END_FUNCTION_BLOCK

// ---- PLC/MAIN.TcPOU
PROGRAM MAIN
VAR
	GetTime: NT_GetTime;
	cpuusage:TC_CpuUsage;
	getLocalAMS: FB_GetLocalAmsNetId;
	ReadSystemInfo:PLC_ReadSymInfo;
	getLatency:TC_SysLatency;
	restartTC:TC_Restart;
	stopTC:TC_Stop;
	configModeTC:TC_Config;
	reqHostName:FB_GetHostName;
	getNetworkadaptors:FB_GetAdaptersInfo;
	getDeviceInfoEx:FB_GetDeviceIdentificationEx;
	
	getLicences:FB_GetLicensesEx;
	
	
	

	oneSec: fb_flasher;
	twoSec: fb_flasher;
	tenSec: fb_flasher;
	oneMSec: fb_flasher;
	hundredMSec: fb_flasher;
	
	pulseoneSec: R_TRIG;
	pulsetwoSec: R_TRIG;
	pulsetenSec: R_TRIG;
	pulseoneMSec: R_TRIG;
	pulsehundredMSec: R_TRIG;
	i: INT;
	nLicPres: UDINT;
	
	oneSecStart:TON;
	
END_VAR

//call PLC data
actPLC();

//call init data for machine
actInit();

//call clock memory
actClockMemory();

//call all diagnostics
actDiag();

//call licence view
actLicenceView();

//call safety main
prgSafetyMain();


//call base machine

//call HMI
//calls logic to drive the HMI
pouHMI();

//call machine base
pouMachine();

//call station 1
//calls motions only associated with station 1
IF System.gSetup.stationEnable[1] THEN pouStation1(); END_IF;

//call station 2
IF System.gSetup.stationEnable[2] THEN pouStation2(); END_IF;

//call station 3
IF System.gSetup.stationEnable[3] THEN pouStation3(); END_IF;

//call station 4
IF System.gSetup.stationEnable[4] THEN pouStation4(); END_IF;

//call station 5
IF System.gSetup.stationEnable[5] THEN pouStation5(); END_IF;

//call station 6
IF System.gSetup.stationEnable[6] THEN pouStation6(); END_IF;

//there are only ever 6 maximum stations

//call logic after station calls for scan after the call of stations
prgAfterStationScan();


//test call for data view
pouDataDisplay();

//call mode rows - call after to use scan logic
prgModeRows();

//call program for machine settings
pouMachineSettings();

//test call for data analyse
prgDataAnaylse();

ACTION actClockMemory:
//clock memory call

//timer call
oneMsec(timeVal:=T#1MS);
System.oneMilliSecond:=oneMSec.q;
pulseoneMSec(CLK:= System.oneMilliSecond);
System.PulseOneMilliSecond := pulseoneMSec.Q;

oneSec(timeVal:=T#1S);
System.OneSecond:=oneSec.q;
pulseoneSec(CLK:= System.OneSecond);
System.PulseOneSecond  := pulseoneSec.Q;

twoSec(timeVal:=T#1S);
System.TwoSecond:=twoSec.q;
pulseTwoSec(CLK:= System.TwoSecond);
System.PulseTwosecond  := pulsetwoSec.Q;

tenSec(timeVal:=T#10S);
System.TenSecond:=tenSec.q;
pulsetenSec(CLK:= System.TenSecond);
System.PulseTenSecond := pulsetenSec.Q;

hundredMSec(timeVal:=T#100MS);
System.hundredMilliSecond:=hundredMSec.q;
pulsehundredMSec(CLK:= System.hundredMilliSecond);
System.PulseHundredMilliSecond := pulsehundredMSec.Q;

oneSecStart(IN:=TRUE);
System.StartPulse:=(oneSecStart.Q);




IF system.thetime.wDay = 28 AND System.thetime.wMonth = 11 THEN
	System.gHappyBirthday := TRUE;
	ELSE
	System.gHappyBirthday := FALSE;
END_IF
END_ACTION

ACTION actDiag:
//call diag blocks
pouDPDiag();
pouEtherCATdiag();
pouPROFINETdiag();
END_ACTION

ACTION actInit:
//block must be called first in scan

//Initalise PLC data for first scan

//activate the first station
IF System.myPlcInfoTask1.FirstCycle THEN
	gHMIData.gActiveStationNumber := 1;
	gHMIData.gStationSelected[1] := TRUE;
	gHMIData.gStationSelected[2] := FALSE;
	gHMIData.gStationSelected[3] := FALSE;
	gHMIData.gStationSelected[4] := FALSE;
	gHMIData.gStationSelected[5] := FALSE;
	gHMIData.gStationSelected[6] := FALSE;
	
	
	//start in manual mode
	S1_Global.station.Data.Manual := TRUE;
	S1_Global.station.Data.AutoCycle := FALSE;
	S1_Global.station.Data.ContCycle := TRUE;
	S1_Global.station.Data.SingleCycle := FALSE;
	
	FC_S1_AssignTaskTimes(iqPartData:=S1_Global.station);
	FC_S2_AssignTaskTimes(iqPartData:=S2_Global.station);
	FC_S3_AssignTaskTimes(iqPartData:=S3_Global.station);
	FC_S4_AssignTaskTimes(iqPartData:=S4_Global.station);
	FC_S5_AssignTaskTimes(iqPartData:=S5_Global.station);
	FC_S6_AssignTaskTimes(iqPartData:=S6_Global.station);
	
	
END_IF

//globals used in future scan(s)
GlobalMessages.gAnyWarnings := FALSE;
GlobalMessages.gAnyFaultMessage := FALSE;

//set other parameters
FC_Setup();
END_ACTION

ACTION actLicenceView:
	//get licence info
	getLicences		(	bExecute:= gLicenceView.tCallUpdateLicenceList,
						tTimeout:=T#10S,
						sNetId:=
					);
	//reset read BOOL
	gLicenceView.tCallUpdateLicenceList := FALSE;
					
gLicenceView.nValidLicences		:=	getLicences.nValidLicenses;
gLicenceView.aValidLicences		:=	getLicences.aValidLicenses;

gLicenceView.nPendingLicences	:=	getLicences.nPendingLicenses;
gLicenceView.aPendingLicences	:=	getLicences.aPendingLicenses;

gLicenceView.nDemoLicences		:=	getLicences.nDemoLicenses;
gLicenceView.aDemoLicences		:=	getLicences.aDemoLicenses;

gLicenceView.nOEMLicences		:=	getLicences.nOemLicenses;
gLicenceView.aOEMLicences		:=	getLicences.aOemLicenses;

gLicenceView.nFailedLicences	:=	getLicences.nFailedLicenses;
gLicenceView.aFailedLicences	:=	getLicences.aFailedLicenses;

gLicenceView.nInvalidLicences	:=	getLicences.nInvalidLicenses;
gLicenceView.aInvalidLicences	:=	getLicences.aInvalidLicenses;

//gLicenceView.maxlicenceIndex := 	gLicenceView.nDemoLicences;
//gLicenceView.tActiveLicenceArray := gLicenceView.ademoLicences[1];


//check if last radio index was changed
IF gLicenceView.licenceType = gLicenceView.tActiveLicenceSelLast THEN
	;
	ELSE
		
	//update list BOOL
	gLicenceView.tCallUpdateLicenceList := TRUE;
	//reset check for next scan
	gLicenceView.tActiveLicenceSelLast :=  gLicenceView.licenceType;
	
END_IF

//assign licence name into array
IF gLicenceView.tCallUpdateLicenceList THEN
	
	//set integer limits for array selection
gLicenceView.tActiveLicenceSel := MAX(gLicenceView.tActiveLicenceSel,1);
gLicenceView.tActiveLicenceSel := MIN(gLicenceView.tActiveLicenceSel,nMaxLicenses);

	
	memset( destAddr:=	ADR(gLicenceView.tActiveLicenceArray),
		 	fillByte:=	16#0,
			n:=			SIZEOF(gLicenceView.tActiveLicenceArray)
			);
	
	memset( destAddr:=	ADR(gLicenceView.tActiveLicenceList),
		 	fillByte:=	16#0,
			n:=			SIZEOF(gLicenceView.tActiveLicenceList)
			);
			
		
	
	
	CASE gLicenceView.licenceType OF
		0:
		gLicenceView.maxlicenceIndex := 	gLicenceView.nValidLicences;
		FOR nLicPres := 1 TO gLicenceView.maxlicenceIndex DO
			gLicenceView.tActiveLicenceList[nLicPres] := gLicenceView.aValidLicences[nLicPres].sLicenseName;
		END_FOR
		
		1:
		gLicenceView.maxlicenceIndex := 	gLicenceView.nPendingLicences;
		FOR nLicPres := 1 TO gLicenceView.maxlicenceIndex DO
			gLicenceView.tActiveLicenceList[nLicPres] := gLicenceView.aPendingLicences[nLicPres].sLicenseName;
		END_FOR
		
		2:
		gLicenceView.maxlicenceIndex := 	gLicenceView.nDemoLicences;
		FOR nLicPres := 1 TO gLicenceView.maxlicenceIndex DO
			gLicenceView.tActiveLicenceList[nLicPres] := gLicenceView.aDemoLicences[nLicPres].sLicenseName;
		END_FOR
		
		3:
		gLicenceView.maxlicenceIndex := 	gLicenceView.nOEMLicences;
		FOR nLicPres := 1 TO gLicenceView.maxlicenceIndex DO
			gLicenceView.tActiveLicenceList[nLicPres] := gLicenceView.aOEMLicences[nLicPres].sLicenseName;
		END_FOR
		
		4:
		gLicenceView.maxlicenceIndex := 	gLicenceView.nFailedLicences;
		FOR nLicPres := 1 TO gLicenceView.maxlicenceIndex DO
			gLicenceView.tActiveLicenceList[nLicPres] := gLicenceView.aFailedLicences[nLicPres].sLicenseName;
		END_FOR
		
		5:
		gLicenceView.maxlicenceIndex := 	gLicenceView.nInvalidLicences;
		FOR nLicPres := 1 TO gLicenceView.maxlicenceIndex DO
			gLicenceView.tActiveLicenceList[nLicPres] := gLicenceView.aInvalidLicences[nLicPres].sLicenseName;
		END_FOR
	
	END_CASE
END_IF

//move data structure into sole struct on HMI
IF gLicenceView.licenceType > 0 THEN

CASE gLicenceView.licenceType OF
	0: 
	//move selected array into viewing arrayh
	gLicenceView.tActiveLicenceArray := gLicenceView.aValidLicences[gLicenceView.tActiveLicenceSel];
	
	1: 
	//move selected array into viewing arrayh
	gLicenceView.tActiveLicenceArray := gLicenceView.aPendingLicences[gLicenceView.tActiveLicenceSel];
	
	2: 
	//move selected array into viewing arrayh
	gLicenceView.tActiveLicenceArray := gLicenceView.aDemoLicences[gLicenceView.tActiveLicenceSel];
	
	3: 
	//move selected array into viewing arrayh
	gLicenceView.tActiveLicenceArray := gLicenceView.aOEMLicences[gLicenceView.tActiveLicenceSel];
	
	4: 
	//move selected array into viewing arrayh
	gLicenceView.tActiveLicenceArray := gLicenceView.aFailedLicences[gLicenceView.tActiveLicenceSel];
	
	5: 
	//move selected array into viewing arrayh
	gLicenceView.tActiveLicenceArray := gLicenceView.aInvalidLicences[gLicenceView.tActiveLicenceSel];
	
END_CASE
END_IF
END_ACTION

ACTION actPLC:
//act call PLC
//get PLC app data
	System.myPlcAppSystemInfo:=TwinCAT_SystemInfoVarList._AppInfo;
	
	//get task info
	System.myPlcInfoTask1 := TwinCAT_SystemInfoVarList._TaskInfo[1];
	
	//move task scan time to memory
	System.ScanTimeReq := UDINT_TO_REAL(System.myPlcInfoTask1.CycleTime);
	System.ScanTimeAct := UDINT_TO_REAL(System.myPlcInfoTask1.LastExecTime);
	
	//scale to correct factor
	System.ScanTimeReq := System.ScanTimeReq / 10000;
	System.ScanTimeAct := System.ScanTimeAct / 10000;
	
	//if the scan time is a new record, then save the scan time and the scan number
	IF System.ScanTimeAct > System.ScanTimeRecord  THEN
		//debug message for new record scan
		System.ScanTimeRecord := System.ScanTimeAct;
		System.ScanTimeRecordScan:= System.myPlcInfoTask1.CycleCount;
	END_IF
	
	//get the local AMS address
	getLocalAMS(	bExecute:=System.myPlcInfoTask1.FirstCycle, 
					tTimeOut:=T#1M
				);
	
	System.AmsNetIdstr:=getLocalAMS.AddrString;
	System.AmsNetIdbytes:=getLocalAMS.AddrBytes;
	
	//get the time
	GetTime(		NETID:='',
					START:=System.OneSecond,
			);
	
	System.thetime:= GetTime.TIMESTR;
	
	//convert timestruct to DT time
	System.timeDT := SYSTEMTIME_TO_DT(TIMESTR:=system.thetime);

	
	//get CPU usage
	cpuusage(	netID:=,
				Start:=System.PulseHundredMilliSecond,
				TMOUT:=T#10S
				);
	System.cpuusageval  := cpuusage.USAGE;
	
	//get symbol count, usage
	ReadSystemInfo( NETID:=,
					Port:=System.myPlcAppSystemInfo.AdsPort,
					Start:=system.OneSecond,
					TMOUT:=T#10S,
					);
	system.symCount:=ReadSystemInfo.SYMCOUNT;
	system.sysSize:=ReadSystemInfo.SYMSIZE;
	
	//get latency
	getLatency(		NETID:=,
					Start:=system.OneSecond,
					TMOUT:=T#10S,
					);
	System.LatencyMicroSec := getLatency.ACTUAL;
	system.MaxLatencyMicroSec := getLatency.MAXIMUM;
	
	//restart TC
	restartTC(		NETID:=,
					Restart:=System.TCRestartReq,
					TMOUT:=T#10S
					);
					
	//stop TC
	stopTC(			NETID:=,
					STOP:=System.TCStopReq,
					TMOUT:=T#10S
					);
					
	//config mode TC
	configModeTC(	NETID:=,
					SET:=System.TCConfigReq,
					TMOUT:=T#10S
					);
				
	//get host name
	reqHostName(	sNetID:=,
					bExecute:=system.TenSecond,
					tTimeout:=T#10S
					);
	System.NThostname := reqHostName.sHostName;
	
	
	//get networkadaptors
	getNetworkadaptors(	sNetID:=,
						bExecute:=system.TenSecond,
						tTimeout:=T#10S,
						);
	System.networkadaptors:=getNetworkadaptors.arrAdapters;
	
	//get Device Infomation
	getDeviceInfoEx(	bExecute := System.sysDeviceUpdate,
						tTimeout := T#10S,
						sNetId:=
					);
					
	System.sysDeviceInfo := getDeviceInfoEx.stDevIdent;
	
	IF gHMIButtons.gAnyMotionButtonPresed THEN gHMIButtons.gAnyMotionButtonPresed := FALSE; END_IF//first scan
END_ACTION

END_PROGRAM

// ---- PLC/FBs/FBs/FB_Flasher.TcPOU
FUNCTION_BLOCK FB_Flasher
VAR
	timON: TON;
	timOFF: TON;

END_VAR

VAR_INPUT
	timeVal:TIME;
	
END_VAR

VAR_OUTPUT
	q:BOOL;

END_VAR

//time on flasher
timON(	IN:= NOT timOFF.Q,
		PT:= timeVal
		);
		
q:= timON.Q;


//time off
timOFF(	IN:= timON.Q,
		PT:= timeVal
		);

END_FUNCTION_BLOCK

// ---- PLC/Safety/prgSafetyMain.TcPOU
PROGRAM prgSafetyMain
VAR
	allowpendantUsage: BOOL; //TRUE if the operator has selected on the HMI to enable the pendant
	runSafeProgram: BOOL; //TRUE to run the safety program
END_VAR



//theme:lOkFAHbeCio

//Main Safety Program Call

//run safety program
IF gHMIButtons.btnReset THEN
	runSafeProgram := TRUE;
END_IF

//add logic TBD to stop safety program

//this send the enable to run the program, should be running all the time in most cases
IF runSafeProgram THEN
	Safety.qInRun := TRUE;
END_IF


//enable pendent logic tbd
allowpendantUsage := FALSE;


//send reset to safety program runtime
IF gHMIButtons.btnReset THEN
	Safety.iResetFBs := TRUE;
	ELSE
	Safety.iResetFBs := FALSE;
END_IF

//to prevent a reset button enabling power devices, have seperate enable fed from HMI
//scan in 0 value
Safety.iEnableSafetyDevicesuint := 0;
IF S1_Global.station.Data.MotionPowerOn AND NOT allowpendantUsage THEN
	//if the station power (or machine power to edit) is on, send value of 1 to enable logic in safety program
	Safety.iEnableSafetyDevicesuint := 1;
END_IF

//pendent enable usage
//scan in 0 value
Safety.iEnablePendantSafetyDevicesuint := 0;
IF allowpendantUsage THEN
	//if the HMI has selected a pendant to use then turn on logic in program
	Safety.iEnablePendantSafetyDevicesuint := 1;
END_IF

END_PROGRAM

// ---- HMI1/Logic/pouHMI.TcPOU
PROGRAM pouHMI
VAR
END_VAR

//all logic to control HMI
prgHMIcontrol();

//control Unit Screen
prgHMIUnits();

//logic for stations
prgHMIstations();

//call to read text lists into PLC memory arrays
prgReadTextList();

//control language Screen
prgHMILanguage();

//axis telegram diag screen
prgHMIaxis();

//lock station logic
actLockStation();

//for Toast-hmi only
actMoveToastHMIData();

ACTION actLockStation:
//lock stations together feedback

IF gHMIButtons.btnLockStation1 THEN gHMIData.gStateLockStation1 := 1; ELSE gHMIData.gStateLockStation1 := 0 ; END_IF
IF gHMIButtons.btnLockStation2 THEN gHMIData.gStateLockStation2 := 1; ELSE gHMIData.gStateLockStation2 := 0 ; END_IF
IF gHMIButtons.btnLockStation3 THEN gHMIData.gStateLockStation3 := 1; ELSE gHMIData.gStateLockStation3 := 0 ; END_IF	
IF gHMIButtons.btnLockStation4 THEN gHMIData.gStateLockStation4 := 1; ELSE gHMIData.gStateLockStation4 := 0 ; END_IF
IF gHMIButtons.btnLockStation5 THEN gHMIData.gStateLockStation5 := 1; ELSE gHMIData.gStateLockStation5 := 0 ; END_IF
IF gHMIButtons.btnLockStation6 THEN gHMIData.gStateLockStation6 := 1; ELSE gHMIData.gStateLockStation6 := 0 ; END_IF
	

//apply locks to stations
S1_Global.station.Data.IsStationLocked	:=	gHMIButtons.btnLockStation1;
S2_Global.station.Data.IsStationLocked	:=	gHMIButtons.btnLockStation2;
S3_Global.station.Data.IsStationLocked	:=	gHMIButtons.btnLockStation3;
S4_Global.station.Data.IsStationLocked	:=	gHMIButtons.btnLockStation4;
S5_Global.station.Data.IsStationLocked	:=	gHMIButtons.btnLockStation5;
S6_Global.station.Data.IsStationLocked	:=	gHMIButtons.btnLockStation6;
END_ACTION

ACTION actMoveToastHMIData:
//move data to new gMHIData to read, not the root for ADS reads

//station selected as BOOL
	gTOASTHMI.gData.hmi.gStationSelected := gHMIData.gStationSelected;
	
	//hide display elements
		gTOASTHMI.gData.hmi.gHideDisplayElements := gHMIData.gHideDisplayElements;
	
	//stations enabled
		gTOASTHMI.gData.hmi.gStationEnabled := gHMIData.gStationEnabled;
	
		gTOASTHMI.gData.hmi.gRowElementOffset := gHMIData.gRowElementOffset;
	
	//number of the active station for message display
		gTOASTHMI.gData.hmi.gNumActivePromptTextList := gHMIData.gNumActivePromptTextList;
		gTOASTHMI.gData.hmi.gNumActiveWarningTextList := gHMIData.gNumActiveWarningTextList;
		gTOASTHMI.gData.hmi.gNumActiveAlarmTextList := gHMIData.gNumActiveAlarmTextList;
	
	//station selected as integer
		gTOASTHMI.gData.hmi.gActiveStationNumber := gHMIData.gActiveStationNumber;
	
		gTOASTHMI.gData.hmi.gActivePageNumber := gHMIData.gActivePageNumber;
		gTOASTHMI.gData.hmi.gMaxPageNumber := gHMIData.gMaxPageNumber;
	
		gTOASTHMI.gData.hmi.gActiveScreen := gHMIData.gActiveScreen;
	
	//machine prompt number to display (summation)
		gTOASTHMI.gData.hmi.gMachinePromptNumber := gHMIData.gMachinePromptNumber;

	//current number of screen on HMI
		gTOASTHMI.gData.hmi.gScreenNumber := gHMIData.gScreenNumber;

	//hide display elements based on what station is selected
		gTOASTHMI.gData.hmi.gHideDisplayElementAlarmView := gHMIData.gHideDisplayElementAlarmView;
		gTOASTHMI.gData.hmi.gHideDisplayElementWarningView := gHMIData.gHideDisplayElementWarningView;
		gTOASTHMI.gData.hmi.gHideDisplayElementPromptView := gHMIData.gHideDisplayElementPromptView;
	
	
		gTOASTHMI.gData.hmi.gAlarmViewMsg := gHMIData.gAlarmViewMsg;
	
	//header data
		gTOASTHMI.gData.hmi.hmiHeader := gHMIData.hmiHeader;
	
	//language screen
		gTOASTHMI.gData.hmi.gLangRowElementOffset := gHMIData.gLangRowElementOffset;
		gTOASTHMI.gData.hmi.gLangRows := gHMIData.gLangRows;
		gTOASTHMI.gData.hmi.gLangButtons := gHMIData.gLangButtons;
		gTOASTHMI.gData.hmi.gActiveLangPageNumber := gHMIData.gActiveLangPageNumber;
		gTOASTHMI.gData.hmi.gMaxPageNumberLang := gHMIData.gMaxPageNumberLang;
	
		gTOASTHMI.gData.hmi.gHMIScreenString := gHMIData.gHMIScreenString;
	
	//title of manual motion screen
		gTOASTHMI.gData.hmi.gManualScreenTitle := gHMIData.gManualScreenTitle;
	
		gTOASTHMI.gData.hmi.gVisuHasInited := gHMIData.gVisuHasInited;
	
	//buttons to lock a station
		gTOASTHMI.gData.hmi.gStateLockStation1 := gHMIData.gStateLockStation1;
		gTOASTHMI.gData.hmi.gStateLockStation2 := gHMIData.gStateLockStation2;
		gTOASTHMI.gData.hmi.gStateLockStation3 := gHMIData.gStateLockStation3;
		gTOASTHMI.gData.hmi.gStateLockStation4 := gHMIData.gStateLockStation4;
		gTOASTHMI.gData.hmi.gStateLockStation5 := gHMIData.gStateLockStation5;
		gTOASTHMI.gData.hmi.gStateLockStation6 := gHMIData.gStateLockStation6;
		
		//////////////////////////
		
		
			//buttons to select a station
	gTOASTHMI.gData.btns.btnSelectStation1 := gHMIButtons.btnSelectStation1;
		gTOASTHMI.gData.btns.btnSelectStation2 := gHMIButtons.btnSelectStation2;
		gTOASTHMI.gData.btns.btnSelectStation3 := gHMIButtons.btnSelectStation3;
		gTOASTHMI.gData.btns.btnSelectStation4 := gHMIButtons.btnSelectStation4;
		gTOASTHMI.gData.btns.btnSelectStation5 := gHMIButtons.btnSelectStation5;
		gTOASTHMI.gData.btns.btnSelectStation6 := gHMIButtons.btnSelectStation6;

		gTOASTHMI.gData.btns.btnSelectAll := gHMIButtons.btnSelectAll;	//button to select all stations
		gTOASTHMI.gData.btns.btnAllStationsSelected := gHMIButtons.btnAllStationsSelected;

	//reset button for global use
		gTOASTHMI.gData.btns.btnReset := gHMIButtons.btnReset;

	//manual screen
		gTOASTHMI.gData.btns.btnAbsMode := gHMIButtons.btnAbsMode; //TRUE if abs mode, False if sys mode
		gTOASTHMI.gData.btns.btnNextPage := gHMIButtons.btnNextPage;
		gTOASTHMI.gData.btns.btnPrevPage := gHMIButtons.btnPrevPage;
	
	//hide button data for main screen
		gTOASTHMI.gData.btns.btnHides := gHMIButtons.btnHides;
	
	//hmi buttons
		gTOASTHMI.gData.btns.btnMode := gHMIButtons.btnMode;
	
	//hmi buttons feedback
		gTOASTHMI.gData.btns.btnFdbk := gHMIButtons.btnFdbk;
	
		gTOASTHMI.gData.btns.btnPlus1Row := gHMIButtons.btnPlus1Row; //scroll 1 row up
		gTOASTHMI.gData.btns.btnNeg1Row := gHMIButtons.btnNeg1Row; //scroll 1 row down
		gTOASTHMI.gData.btns.clk := gHMIButtons.clk;
	
		gTOASTHMI.gData.btns.gAnyButtonPressed := 	gHMIButtons.gAnyButtonPressed; //TRUE if any button was pressed
	
		//buttons to lock a station
		gTOASTHMI.gData.btns.btnLockStation1 := gHMIButtons.btnLockStation1;
		gTOASTHMI.gData.btns.btnLockStation2 := gHMIButtons.btnLockStation2;
		gTOASTHMI.gData.btns.btnLockStation3 := gHMIButtons.btnLockStation3;
		gTOASTHMI.gData.btns.btnLockStation4 := gHMIButtons.btnLockStation4;
		gTOASTHMI.gData.btns.btnLockStation5 := gHMIButtons.btnLockStation5;
		gTOASTHMI.gData.btns.btnLockStation6 := gHMIButtons.btnLockStation6;
	
		gTOASTHMI.gData.btns.gLockButtons := gHMIButtons.gLockButtons;
		
		
		//move messages
		
		gTOASTHMI.gData.GlobalMessages.gMsgMc	:= GlobalMessages.gMsgMc;
	
	//define message for each station
	gTOASTHMI.gData.GlobalMessages.gMsgS1		:= GlobalMessages.gMsgS1;
	gTOASTHMI.gData.GlobalMessages.gMsgS2		:= GlobalMessages.gMsgS2;
	gTOASTHMI.gData.GlobalMessages.gMsgS3		:= GlobalMessages.gMsgS3;
	gTOASTHMI.gData.GlobalMessages.gMsgS4		:= GlobalMessages.gMsgS4;
	gTOASTHMI.gData.GlobalMessages.gMsgS5		:= GlobalMessages.gMsgS5;
	gTOASTHMI.gData.GlobalMessages.gMsgS6		:= GlobalMessages.gMsgS6;
	
	//global memory for retaining status of station
	gTOASTHMI.gData.GlobalMessages.gMsgMcStat		:= GlobalMessages.gMsgMcStat;
	gTOASTHMI.gData.GlobalMessages.gMsgS1Stat		:= GlobalMessages.gMsgS1Stat;
	gTOASTHMI.gData.GlobalMessages.gMsgS2Stat		:= GlobalMessages.gMsgS2Stat;
	gTOASTHMI.gData.GlobalMessages.gMsgS3Stat		:= GlobalMessages.gMsgS3Stat;
	gTOASTHMI.gData.GlobalMessages.gMsgS4Stat		:= GlobalMessages.gMsgS4Stat;
	gTOASTHMI.gData.GlobalMessages.gMsgS5Stat		:= GlobalMessages.gMsgS5Stat;
	gTOASTHMI.gData.GlobalMessages.gMsgS6Stat		:= GlobalMessages.gMsgS6Stat;
	
	//list view of messages in array form
	gTOASTHMI.gData.GlobalMessages.gListMsgMc		:= GlobalMessages.gListMsgMc;
	gTOASTHMI.gData.GlobalMessages.gListMsgS1		:= GlobalMessages.gListMsgS1;
	gTOASTHMI.gData.GlobalMessages.gListMsgS2		:= GlobalMessages.gListMsgS2;
	gTOASTHMI.gData.GlobalMessages.gListMsgS3		:= GlobalMessages.gListMsgS3;
	gTOASTHMI.gData.GlobalMessages.gListMsgS4		:= GlobalMessages.gListMsgS4;
	gTOASTHMI.gData.GlobalMessages.gListMsgS5		:= GlobalMessages.gListMsgS5;
	gTOASTHMI.gData.GlobalMessages.gListMsgS6		:= GlobalMessages.gListMsgS6;

	gTOASTHMI.gData.GlobalMessages.gAnyFaultMessage	:= GlobalMessages.gAnyFaultMessage; //TRUE if there are any fault messages (any)
	gTOASTHMI.gData.GlobalMessages.gAnyWarnings	:= GlobalMessages.gAnyWarnings; //TRUE if there are any warnings (the yellow ones)

	//alarm view of messages in alarmview form
	gTOASTHMI.gData.GlobalMessages.gMcAlarmView	:= GlobalMessages.gMcAlarmView;
	gTOASTHMI.gData.GlobalMessages.gS1AlarmView	:= GlobalMessages.gS1AlarmView;
	gTOASTHMI.gData.GlobalMessages.gS2AlarmView	:= GlobalMessages.gS2AlarmView;
	gTOASTHMI.gData.GlobalMessages.gS3AlarmView	:= GlobalMessages.gS3AlarmView;
	gTOASTHMI.gData.GlobalMessages.gS4AlarmView	:= GlobalMessages.gS4AlarmView;
	gTOASTHMI.gData.GlobalMessages.gS5AlarmView	:= GlobalMessages.gS5AlarmView;
	gTOASTHMI.gData.GlobalMessages.gS6AlarmView	:= GlobalMessages.gS6AlarmView;
	
	gTOASTHMI.gData.GlobalMessages.gHMIAlarmView	:= GlobalMessages.gHMIAlarmView;
END_ACTION

ACTION actResetButtonPress:
//if its on, then turn it off, it will be taken in other places
IF gHMIButtons.gAnyButtonPressed AND System.PulseTenSecond THEN
	gHMIButtons.gAnyButtonPressed := FALSE;
END_IF
END_ACTION

END_PROGRAM

// ---- HMI1/Logic/prgHMIcontrol.TcPOU
PROGRAM prgHMIcontrol
VAR
	retval: UDINT;
	retvalll: UDINT;
	a: INT;
	workString: STRING(255);
	strLen: INT;
	b: INT;
	workString2: STRING(255);
	c: INT;
END_VAR

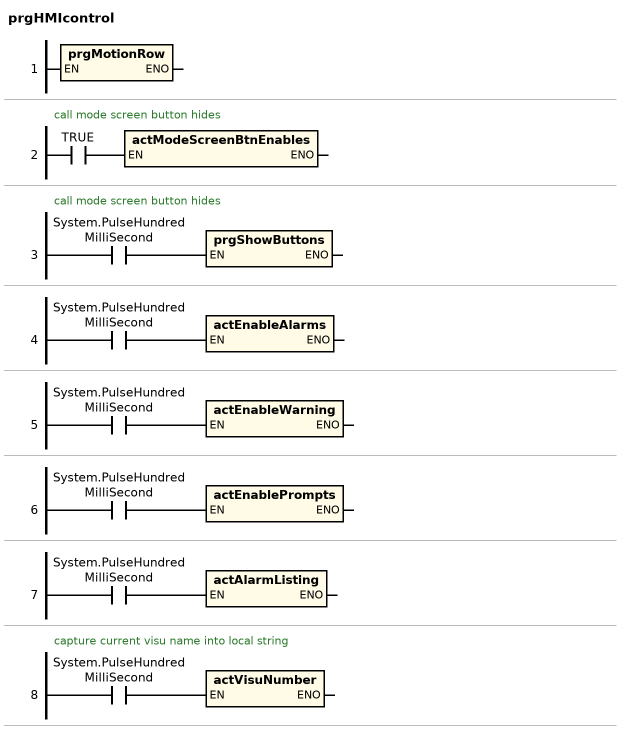
// NETWORK 1
prgMotionRow();

// NETWORK 2
// call mode screen button hides
actModeScreenBtnEnables();

// NETWORK 3
// call mode screen button hides
IF System.PulseHundredMilliSecond THEN prgShowButtons(); END_IF

// NETWORK 4
IF System.PulseHundredMilliSecond THEN actEnableAlarms(); END_IF

// NETWORK 5
IF System.PulseHundredMilliSecond THEN actEnableWarning(); END_IF

// NETWORK 6
IF System.PulseHundredMilliSecond THEN actEnablePrompts(); END_IF

// NETWORK 7
IF System.PulseHundredMilliSecond THEN actAlarmListing(); END_IF

// NETWORK 8
// capture current visu name into local string
IF System.PulseHundredMilliSecond THEN actVisuNumber(); END_IF

ACTION actAlarmListing:
//do nothing


//do something
//move station data into global data area for viewing
IF gHMIData.gStationSelected[1] THEN
	retvalll := MEMCPY(	destAddr:=	ADR(	gHMIData.gAlarmViewMsg), 
						srcAddr:=	ADR(	GlobalMessages.gListMsgS1), 
						n:=			SIZEOF(	GlobalMessages.gListMsgS1));
						
	retvalll := MEMCPY(	destAddr:=	ADR(	GlobalMessages.gHMIAlarmView), 
						srcAddr:=	ADR(	GlobalMessages.gS1AlarmView), 
						n:=			SIZEOF(	GlobalMessages.gS1AlarmView));
END_IF

IF gHMIData.gStationSelected[2] THEN
	retvalll := MEMCPY(	destAddr:=	ADR(	gHMIData.gAlarmViewMsg), 
						srcAddr:=	ADR(	GlobalMessages.gListMsgS2), 
						n:=			SIZEOF(	GlobalMessages.gListMsgS2));
						
	retvalll := MEMCPY(	destAddr:=	ADR(	GlobalMessages.gHMIAlarmView), 
						srcAddr:=	ADR(	GlobalMessages.gS2AlarmView), 
						n:=			SIZEOF(	GlobalMessages.gS2AlarmView));
END_IF

IF gHMIData.gStationSelected[3] THEN
	retvalll := MEMCPY(	destAddr:=	ADR(	gHMIData.gAlarmViewMsg), 
						srcAddr:=	ADR(	GlobalMessages.gListMsgS3), 
						n:=			SIZEOF(	GlobalMessages.gListMsgS3));

	retvalll := MEMCPY(	destAddr:=	ADR(	GlobalMessages.gHMIAlarmView), 
						srcAddr:=	ADR(	GlobalMessages.gS3AlarmView), 
						n:=			SIZEOF(	GlobalMessages.gS3AlarmView));
END_IF

IF gHMIData.gStationSelected[4] THEN
	retvalll := MEMCPY(	destAddr:=	ADR(	gHMIData.gAlarmViewMsg), 
						srcAddr:=	ADR(	GlobalMessages.gListMsgS4), 
						n:=			SIZEOF(	GlobalMessages.gListMsgS4));

	retvalll := MEMCPY(	destAddr:=	ADR(	GlobalMessages.gHMIAlarmView), 
						srcAddr:=	ADR(	GlobalMessages.gS4AlarmView), 
						n:=			SIZEOF(	GlobalMessages.gS4AlarmView));
END_IF

IF gHMIData.gStationSelected[5] THEN
	retvalll := MEMCPY(	destAddr:=	ADR(	gHMIData.gAlarmViewMsg), 
						srcAddr:=	ADR(	GlobalMessages.gListMsgS5), 
						n:=			SIZEOF(	GlobalMessages.gListMsgS5));

	retvalll := MEMCPY(	destAddr:=	ADR(	GlobalMessages.gHMIAlarmView), 
						srcAddr:=	ADR(	GlobalMessages.gS5AlarmView), 
						n:=			SIZEOF(	GlobalMessages.gS5AlarmView));

END_IF

IF gHMIData.gStationSelected[6] THEN
	retvalll := MEMCPY(	destAddr:=	ADR(	gHMIData.gAlarmViewMsg), 
						srcAddr:=	ADR(	GlobalMessages.gListMsgS6), 
						n:=			SIZEOF(	GlobalMessages.gListMsgS6));

	retvalll := MEMCPY(	destAddr:=	ADR(	GlobalMessages.gHMIAlarmView), 
						srcAddr:=	ADR(	GlobalMessages.gS6AlarmView), 
						n:=			SIZEOF(	GlobalMessages.gS6AlarmView));
END_IF
END_ACTION

ACTION actEnableAlarms:
//enable alarm views on alarm state
IF GlobalMessages.gMsgMcStat.IsAlarm THEN
	gHMIData.gHideDisplayElementAlarmView.McEnabled := FALSE;
ELSE
	gHMIData.gHideDisplayElementAlarmView.McEnabled := TRUE;
END_IF

//1
IF gHMIData.gStationSelected[1] AND GlobalMessages.gMsgS1Stat.IsAlarm AND NOT GlobalMessages.gMsgMcStat.IsAlarm THEN
	gHMIData.gHideDisplayElementAlarmView.S1Enabled := FALSE;
END_IF

IF NOT GlobalMessages.gMsgS1Stat.IsAlarm THEN
	gHMIData.gHideDisplayElementAlarmView.S1Enabled := TRUE;
END_IF

//2
IF gHMIData.gStationSelected[2] AND GlobalMessages.gMsgS2Stat.IsAlarm AND NOT GlobalMessages.gMsgMcStat.IsAlarm THEN
	gHMIData.gHideDisplayElementAlarmView.S2Enabled := FALSE;
END_IF

IF NOT GlobalMessages.gMsgS2Stat.IsAlarm THEN
	gHMIData.gHideDisplayElementAlarmView.S2Enabled := TRUE;
END_IF

//3
IF gHMIData.gStationSelected[3] AND GlobalMessages.gMsgS3Stat.IsAlarm AND NOT GlobalMessages.gMsgMcStat.IsAlarm THEN
	gHMIData.gHideDisplayElementAlarmView.S3Enabled := FALSE;
END_IF

IF NOT GlobalMessages.gMsgS3Stat.IsAlarm THEN
	gHMIData.gHideDisplayElementAlarmView.S3Enabled := TRUE;
END_IF

//4
IF gHMIData.gStationSelected[4] AND GlobalMessages.gMsgS4Stat.IsAlarm AND NOT GlobalMessages.gMsgMcStat.IsAlarm THEN
	gHMIData.gHideDisplayElementAlarmView.S4Enabled := FALSE;
END_IF

IF NOT GlobalMessages.gMsgS4Stat.IsAlarm THEN
	gHMIData.gHideDisplayElementAlarmView.S4Enabled := TRUE;
END_IF

//5
IF gHMIData.gStationSelected[5] AND GlobalMessages.gMsgS5Stat.IsAlarm AND NOT GlobalMessages.gMsgMcStat.IsAlarm THEN
	gHMIData.gHideDisplayElementAlarmView.S5Enabled := FALSE;
END_IF

IF NOT GlobalMessages.gMsgS5Stat.IsAlarm THEN
	gHMIData.gHideDisplayElementAlarmView.S5Enabled := TRUE;
END_IF

//6
IF gHMIData.gStationSelected[6] AND GlobalMessages.gMsgS6Stat.IsAlarm AND NOT GlobalMessages.gMsgMcStat.IsAlarm THEN
	gHMIData.gHideDisplayElementAlarmView.S6Enabled := FALSE;
END_IF

IF NOT GlobalMessages.gMsgS6Stat.IsAlarm THEN
	gHMIData.gHideDisplayElementAlarmView.S6Enabled := TRUE;
END_IF

//move set global fault
IF GlobalMessages.gMsgS1Stat.IsAlarm THEN
	S1_Global.station.Data.Fault := TRUE;
	ELSE
	S1_Global.station.Data.Fault := FALSE;
END_IF

//move set global fault
IF GlobalMessages.gMsgS2Stat.IsAlarm THEN
	S2_Global.station.Data.Fault := TRUE;
	ELSE
	S2_Global.station.Data.Fault := FALSE;
END_IF

//move set global fault
IF GlobalMessages.gMsgS3Stat.IsAlarm THEN
	S3_Global.station.Data.Fault := TRUE;
	ELSE
	S3_Global.station.Data.Fault := FALSE;
END_IF

//move set global fault
IF GlobalMessages.gMsgS4Stat.IsAlarm THEN
	S4_Global.station.Data.Fault := TRUE;
	ELSE
	S4_Global.station.Data.Fault := FALSE;
END_IF

//move set global fault
IF GlobalMessages.gMsgS5Stat.IsAlarm THEN
	S5_Global.station.Data.Fault := TRUE;
	ELSE
	S5_Global.station.Data.Fault := FALSE;
END_IF

//move set global fault
IF GlobalMessages.gMsgS6Stat.IsAlarm THEN
	S6_Global.station.Data.Fault := TRUE;
	ELSE
	S6_Global.station.Data.Fault := FALSE;
END_IF
END_ACTION

ACTION actEnablePrompts:
//enable Prompt views on Prompt state
IF GlobalMessages.gMsgMcStat.IsPrompt THEN
	gHMIData.gHideDisplayElementPromptView.McEnabled := FALSE;
ELSE
	gHMIData.gHideDisplayElementPromptView.McEnabled := TRUE;
END_IF

//1
IF gHMIData.gStationSelected[1] AND GlobalMessages.gMsgS1Stat.IsPrompt THEN
	gHMIData.gHideDisplayElementPromptView.S1Enabled := FALSE;
END_IF

IF NOT GlobalMessages.gMsgS1Stat.IsPrompt THEN
	gHMIData.gHideDisplayElementPromptView.S1Enabled := TRUE;
END_IF

//2
IF gHMIData.gStationSelected[2] AND GlobalMessages.gMsgS2Stat.IsPrompt THEN
	gHMIData.gHideDisplayElementPromptView.S2Enabled := FALSE;
END_IF

IF NOT GlobalMessages.gMsgS2Stat.IsPrompt THEN
	gHMIData.gHideDisplayElementPromptView.S2Enabled := TRUE;
END_IF

//3
IF gHMIData.gStationSelected[3] AND GlobalMessages.gMsgS3Stat.IsPrompt THEN
	gHMIData.gHideDisplayElementPromptView.S3Enabled := FALSE;
END_IF

IF NOT GlobalMessages.gMsgS3Stat.IsPrompt THEN
	gHMIData.gHideDisplayElementPromptView.S3Enabled := TRUE;
END_IF

//4
IF gHMIData.gStationSelected[4] AND GlobalMessages.gMsgS4Stat.IsPrompt THEN
	gHMIData.gHideDisplayElementPromptView.S4Enabled := FALSE;
END_IF

IF NOT GlobalMessages.gMsgS4Stat.IsPrompt THEN
	gHMIData.gHideDisplayElementPromptView.S4Enabled := TRUE;
END_IF

//5
IF gHMIData.gStationSelected[5] AND GlobalMessages.gMsgS5Stat.IsPrompt THEN
	gHMIData.gHideDisplayElementPromptView.S5Enabled := FALSE;
END_IF

IF NOT GlobalMessages.gMsgS5Stat.IsPrompt THEN
	gHMIData.gHideDisplayElementPromptView.S5Enabled := TRUE;
END_IF

//6
IF gHMIData.gStationSelected[6] AND GlobalMessages.gMsgS6Stat.IsPrompt THEN
	gHMIData.gHideDisplayElementPromptView.S6Enabled := FALSE;
END_IF

IF NOT GlobalMessages.gMsgS6Stat.IsPrompt THEN
	gHMIData.gHideDisplayElementPromptView.S6Enabled := TRUE;
END_IF
END_ACTION

ACTION actEnableWarning:
//enable Warning views on Warning state
IF GlobalMessages.gMsgMcStat.IsWarning THEN
	gHMIData.gHideDisplayElementWarningView.McEnabled := FALSE;
ELSE
	gHMIData.gHideDisplayElementWarningView.McEnabled := TRUE;
END_IF

//1
IF gHMIData.gStationSelected[1] AND GlobalMessages.gMsgS1Stat.IsWarning THEN
	gHMIData.gHideDisplayElementWarningView.S1Enabled := FALSE;
END_IF

IF NOT GlobalMessages.gMsgS1Stat.IsWarning THEN
	gHMIData.gHideDisplayElementWarningView.S1Enabled := TRUE;
END_IF

//2
IF gHMIData.gStationSelected[2] AND GlobalMessages.gMsgS2Stat.IsWarning THEN
	gHMIData.gHideDisplayElementWarningView.S2Enabled := FALSE;
END_IF

IF NOT GlobalMessages.gMsgS2Stat.IsWarning THEN
	gHMIData.gHideDisplayElementWarningView.S2Enabled := TRUE;
END_IF

//3
IF gHMIData.gStationSelected[3] AND GlobalMessages.gMsgS3Stat.IsWarning THEN
	gHMIData.gHideDisplayElementWarningView.S3Enabled := FALSE;
END_IF

IF NOT GlobalMessages.gMsgS3Stat.IsWarning THEN
	gHMIData.gHideDisplayElementWarningView.S3Enabled := TRUE;
END_IF

//4
IF gHMIData.gStationSelected[4] AND GlobalMessages.gMsgS4Stat.IsWarning THEN
	gHMIData.gHideDisplayElementWarningView.S4Enabled := FALSE;
END_IF

IF NOT GlobalMessages.gMsgS4Stat.IsWarning THEN
	gHMIData.gHideDisplayElementWarningView.S4Enabled := TRUE;
END_IF

//5
IF gHMIData.gStationSelected[5] AND GlobalMessages.gMsgS5Stat.IsWarning THEN
	gHMIData.gHideDisplayElementWarningView.S5Enabled := FALSE;
END_IF

IF NOT GlobalMessages.gMsgS5Stat.IsWarning THEN
	gHMIData.gHideDisplayElementWarningView.S5Enabled := TRUE;
END_IF

//6
IF gHMIData.gStationSelected[6] AND GlobalMessages.gMsgS6Stat.IsWarning THEN
	gHMIData.gHideDisplayElementWarningView.S6Enabled := FALSE;
END_IF

IF NOT GlobalMessages.gMsgS6Stat.IsWarning THEN
	gHMIData.gHideDisplayElementWarningView.S6Enabled := TRUE;
END_IF


//move set global fault
IF GlobalMessages.gMsgS1Stat.IsWarning THEN
	S1_Global.station.Data.Warning := TRUE;
	ELSE
	S1_Global.station.Data.Warning := FALSE;
END_IF

//move set global fault
IF GlobalMessages.gMsgS2Stat.IsWarning THEN
	S2_Global.station.Data.Warning := TRUE;
	ELSE
	S2_Global.station.Data.Warning := FALSE;
END_IF

//move set global fault
IF GlobalMessages.gMsgS3Stat.IsWarning THEN
	S3_Global.station.Data.Warning := TRUE;
	ELSE
	S3_Global.station.Data.Warning := FALSE;
END_IF

//move set global fault
IF GlobalMessages.gMsgS4Stat.IsWarning THEN
	S4_Global.station.Data.Warning := TRUE;
	ELSE
	S4_Global.station.Data.Warning := FALSE;
END_IF

//move set global fault
IF GlobalMessages.gMsgS5Stat.IsWarning THEN
	S5_Global.station.Data.Warning := TRUE;
	ELSE
	S5_Global.station.Data.Warning := FALSE;
END_IF

//move set global fault
IF GlobalMessages.gMsgS6Stat.IsWarning THEN
	S6_Global.station.Data.Warning := TRUE;
	ELSE
	S6_Global.station.Data.Warning := FALSE;
END_IF
END_ACTION

ACTION actModeScreenBtnEnables:
//theme:LT-b1qXznKI
//hide/show buttons on mode screen

//row 0
gHMIButtons.btnFdbk.btn00Fdbk := FALSE;
gHMIButtons.btnFdbk.btn01Fdbk := FALSE;
gHMIButtons.btnFdbk.btn02Fdbk := FALSE;
gHMIButtons.btnFdbk.btn03Fdbk := FALSE;
gHMIButtons.btnFdbk.btn04Fdbk := FALSE;
gHMIButtons.btnFdbk.btn05Fdbk := FALSE;
gHMIButtons.btnFdbk.btn06Fdbk := FALSE;
gHMIButtons.btnFdbk.btn07Fdbk := FALSE;
gHMIButtons.btnFdbk.btn08Fdbk := FALSE;
gHMIButtons.btnFdbk.btn09Fdbk := FALSE;

//row 1
gHMIButtons.btnFdbk.btn10Fdbk := FALSE;
gHMIButtons.btnFdbk.btn11Fdbk := FALSE;
gHMIButtons.btnFdbk.btn12Fdbk := FALSE;
gHMIButtons.btnFdbk.btn12Fdbk := FALSE;
gHMIButtons.btnFdbk.btn13Fdbk := FALSE;
gHMIButtons.btnFdbk.btn14Fdbk := FALSE;
gHMIButtons.btnFdbk.btn15Fdbk := FALSE;
gHMIButtons.btnFdbk.btn16Fdbk := FALSE;
gHMIButtons.btnFdbk.btn17Fdbk := FALSE;
gHMIButtons.btnFdbk.btn18Fdbk := FALSE;
gHMIButtons.btnFdbk.btn19Fdbk := FALSE;

//row 2
gHMIButtons.btnFdbk.btn20Fdbk := FALSE;
gHMIButtons.btnFdbk.btn21Fdbk := FALSE;
gHMIButtons.btnFdbk.btn22Fdbk := FALSE;
gHMIButtons.btnFdbk.btn22Fdbk := FALSE;
gHMIButtons.btnFdbk.btn23Fdbk := FALSE;
gHMIButtons.btnFdbk.btn24Fdbk := FALSE;
gHMIButtons.btnFdbk.btn25Fdbk := FALSE;
gHMIButtons.btnFdbk.btn26Fdbk := FALSE;
gHMIButtons.btnFdbk.btn27Fdbk := FALSE;
gHMIButtons.btnFdbk.btn28Fdbk := FALSE;
gHMIButtons.btnFdbk.btn29Fdbk := FALSE;

//special row
gHMIButtons.btnFdbk.btnAutoCyclingFdbk := FALSE;
gHMIButtons.btnFdbk.btnIsHomeFdbk := FALSE;
gHMIButtons.btnFdbk.btnModeFdbk := FALSE;
gHMIButtons.btnFdbk.btnIsSEOCFdbk := FALSE;
gHMIButtons.btnFdbk.btnControlFdbk := FALSE;
END_ACTION

ACTION actPartStatus:
//may not need any of this, as the part data is moved to mc_global.part in each part process call
//move station data into global data area for viewing
IF gHMIData.gStationSelected[1] THEN
	retval := memcpy(	destAddr:=	ADR(Mc_Global.part),
						srcAddr:=	ADR(S1_Global.station.part),
						n:=			SIZEOF(S1_Global.station.part)
						);
END_IF

//move station data into global data area for viewing
IF gHMIData.gStationSelected[2] THEN
	retval := memcpy(	destAddr:=	ADR(Mc_Global.part),
						srcAddr:=	ADR(S2_Global.station.part),
						n:=			SIZEOF(S2_Global.station.part)
						);
END_IF

//move station data into global data area for viewing
IF gHMIData.gStationSelected[3] THEN
	retval := memcpy(	destAddr:=	ADR(Mc_Global.part),
						srcAddr:=	ADR(S3_Global.station.part),
						n:=			SIZEOF(S3_Global.station.part)
						);
END_IF

//move station data into global data area for viewing
IF gHMIData.gStationSelected[4] THEN
	retval := memcpy(	destAddr:=	ADR(Mc_Global.part),
						srcAddr:=	ADR(S4_Global.station.part),
						n:=			SIZEOF(S4_Global.station.part)
						);
END_IF

//move station data into global data area for viewing
IF gHMIData.gStationSelected[5] THEN
	retval := memcpy(	destAddr:=	ADR(Mc_Global.part),
						srcAddr:=	ADR(S5_Global.station.part),
						n:=			SIZEOF(S5_Global.station.part)
						);
END_IF

//move station data into global data area for viewing
IF gHMIData.gStationSelected[6] THEN
	retval := memcpy(	destAddr:=	ADR(Mc_Global.part),
						srcAddr:=	ADR(S6_Global.station.part),
						n:=			SIZEOF(S6_Global.station.part)
						);
END_IF
END_ACTION

ACTION actVisuNumber:
//gHMIData.gHMIScreenString
gHMIData.gHMIScreenString := VisuElems.CURRENTVISU;

//get string Leng
strLen:= LEN(STR:=gHMIData.gHMIScreenString);

//find locations
//cut start
a := find(STR1:=gHMIData.gHMIScreenString, STR2:='_');
workString := RIGHT(STR:=gHMIData.gHMIScreenString,size:=strLen - a);

//cut end
b := find(STR1:=workString, STR2:='_');
workString2 := LEFT(STR:=workString,size:=b - 1);


IF a = 0 OR b = 0 THEN
	gHMIData.gScreenNumber := 32767;
	ELSE
	gHMIData.gScreenNumber := STRING_TO_UINT(workString2);
END_IF
END_ACTION

END_PROGRAM

// ---- HMI1/Logic/prgMotionRow.TcPOU
PROGRAM prgMotionRow
VAR
		tStationNumberIndex: UINT;	
		tNumElementsPerScreen: UINT;
		tScreenElementsPerPage: UINT;
		tTrueStationIndex: UINT;
		tSizeOfMotionRow: UINT;
		tSizeOfMotionRowButtons: UINT;
		retval: UDINT;
		btnNext:R_TRIG;
		btnPrev:R_TRIG;
		
		btnNextRow:R_TRIG;
		btnPrevRow:R_TRIG;
		tSingleRowOffset: UINT;
		
	tSingleRowOffsettest: UINT;
	tSingleRowOffsettestbtns: UINT;
	tSizeOfButtonsLen: UINT;
	tSizeOfRowSingleLens: UINT;
	
	tSingleRowOffsetFactor:UINT;
	tSingleRowOffsetPointer: UINT;
END_VAR

//call logic for Motion screen using motion Rows

//select station on HMI
actPageControl();

//calculate screen range
actCalcScreenNumber();

//call manual screen rows
actCallMotionScreen();

//calculate screen range
actCalcMotionRowPosn();

//calculate page title
actCalcPageTitle();

ACTION actCalcMotionRowPosn:
//calaculate station index for pages
tTrueStationIndex := tStationNumberIndex + ((tScreenElementsPerPage * gHMIData.gActivePageNumber) -  tScreenElementsPerPage);


tSingleRowOffsetPointer := (tSingleRowOffsetFactor *  gHMIDataConst.gNumberElementsPerRow) - gHMIDataConst.gNumberElementsPerRow;
tSingleRowOffsetPointer := tSingleRowOffsetPointer + gHMIDataConst.gNumberElementsPerRow;

//test for singular row change
tTrueStationIndex := tTrueStationIndex + tSingleRowOffsetPointer;

//calculate offset for row x
gHMIData.gRowElementOffset[1]:= tTrueStationIndex + ((gHMIDataConst.gNumberElementsPerRow * 1) - gHMIDataConst.gNumberElementsPerRow);
gHMIData.gRowElementOffset[2]:= tTrueStationIndex + ((gHMIDataConst.gNumberElementsPerRow * 2) - gHMIDataConst.gNumberElementsPerRow);
gHMIData.gRowElementOffset[3]:= tTrueStationIndex + ((gHMIDataConst.gNumberElementsPerRow * 3) - gHMIDataConst.gNumberElementsPerRow);
gHMIData.gRowElementOffset[4]:= tTrueStationIndex + ((gHMIDataConst.gNumberElementsPerRow * 4) - gHMIDataConst.gNumberElementsPerRow);
gHMIData.gRowElementOffset[5]:= tTrueStationIndex + ((gHMIDataConst.gNumberElementsPerRow * 5) - gHMIDataConst.gNumberElementsPerRow);
gHMIData.gRowElementOffset[6]:= tTrueStationIndex + ((gHMIDataConst.gNumberElementsPerRow * 6) - gHMIDataConst.gNumberElementsPerRow);
gHMIData.gRowElementOffset[7]:= tTrueStationIndex + ((gHMIDataConst.gNumberElementsPerRow * 7) - gHMIDataConst.gNumberElementsPerRow);
gHMIData.gRowElementOffset[8]:= tTrueStationIndex + ((gHMIDataConst.gNumberElementsPerRow * 8) - gHMIDataConst.gNumberElementsPerRow);
gHMIData.gRowElementOffset[9]:= tTrueStationIndex + ((gHMIDataConst.gNumberElementsPerRow * 9) - gHMIDataConst.gNumberElementsPerRow);


//move to global to be picked up by each row
gHMIMotionRows.gMotionRows.gMotionRow1.IndexLocation := gHMIData.gRowElementOffset[1];
gHMIMotionRows.gMotionRows.gMotionRow2.IndexLocation := gHMIData.gRowElementOffset[2];
gHMIMotionRows.gMotionRows.gMotionRow3.IndexLocation := gHMIData.gRowElementOffset[3];
gHMIMotionRows.gMotionRows.gMotionRow4.IndexLocation := gHMIData.gRowElementOffset[4];
gHMIMotionRows.gMotionRows.gMotionRow5.IndexLocation := gHMIData.gRowElementOffset[5];
gHMIMotionRows.gMotionRows.gMotionRow6.IndexLocation := gHMIData.gRowElementOffset[6];
gHMIMotionRows.gMotionRows.gMotionRow7.IndexLocation := gHMIData.gRowElementOffset[7];
gHMIMotionRows.gMotionRows.gMotionRow8.IndexLocation := gHMIData.gRowElementOffset[8];
gHMIMotionRows.gMotionRows.gMotionRow9.IndexLocation := gHMIData.gRowElementOffset[9];
END_ACTION

ACTION actCalcPageTitle:
//get the page number index relating the group of motions displayed
gHMIData.gManualScreenTitle := tStationNumberIndex + gHMIData.gActivePageNumber;

//10001 = station 1, page 1
//10002 = station 1, page 2

//20001 = station 1, page 1
//etc

//assign text in textlist ManualPageTitle
END_ACTION

ACTION actCalcScreenNumber:
//create number for station
tStationNumberIndex := gHMIData.gActiveStationNumber * 10000;

//calculate number of elements per screen
tNumElementsPerScreen := gHMIDataConst.gNumberRowsPerPage * gHMIDataConst.gNumberElementsPerRow;

//calculate screen per page index
tScreenElementsPerPage := tNumElementsPerScreen  * 1;
END_ACTION

ACTION actCallMotionScreen:
//calculate byte offset - motions
tSizeOfMotionRow		:= gHMIData.gActivePageNumber * SIZEOF(gHMIMotionRows.gMotionRows);
tSizeOfMotionRow 		:= tSizeOfMotionRow - SIZEOF(gHMIMotionRows.gMotionRows);

//test for singular row changes
tSizeOfRowSingleLens := SIZEOF(typeMotionRow); //typ 153 bytes
tSizeOfMotionRow := tSizeOfMotionRow + (tSingleRowOffsetFactor * tSizeOfRowSingleLens) ;


//calculate byte offset - buttons
tSizeOfMotionRowButtons := gHMIData.gActivePageNumber * SIZEOF(gHMIMotionRows.gMotionRowButtons);
tSizeOfMotionRowButtons := tSizeOfMotionRowButtons - SIZEOF(gHMIMotionRows.gMotionRowButtons);

//test for singular row changes
tSizeOfButtonsLen := SIZEOF(typeMotionRowButtons); // typ 83 bytes
tSizeOfMotionRowButtons := tSizeOfMotionRowButtons + (tSingleRowOffsetFactor * tSizeOfButtonsLen);

//move data based on station and page number
//Move feedback indicator data
//Move Button BOOL state back adr(S1_Global.MotionRow)
IF gHMIData.gStationSelected[1] THEN
	retval := memcpy(	destAddr:=	ADR(gHMIMotionRows.gMotionRows),
						srcAddr:=	ADR(S1_Global.station.MotionRow) + tSizeOfMotionRow,
						n:=			SIZEOF(gHMIMotionRows.gMotionRows)
						);
						
	retval := memcpy(	destAddr:=	ADR(S1_Global.station.MotionRowBtn) + tSizeOfMotionRowButtons,
						srcAddr:=	ADR(gHMIMotionRows.gMotionRowButtons),
						n:=			SIZEOF(gHMIMotionRows.gMotionRowButtons)
						);
END_IF

IF gHMIData.gStationSelected[2] THEN
	retval := memcpy(	destAddr:=	ADR(gHMIMotionRows.gMotionRows),
						srcAddr:=	ADR(S2_Global.station.MotionRow) + tSizeOfMotionRow,
						n:=			SIZEOF(gHMIMotionRows.gMotionRows)
						);
						
	retval := memcpy(	destAddr:=	ADR(S2_Global.station.MotionRowBtn) + tSizeOfMotionRowButtons,
						srcAddr:=	ADR(gHMIMotionRows.gMotionRowButtons),
						n:=			SIZEOF(gHMIMotionRows.gMotionRowButtons)
						);
END_IF

IF gHMIData.gStationSelected[3] THEN
	retval := memcpy(	destAddr:=	ADR(gHMIMotionRows.gMotionRows),
						srcAddr:=	ADR(S3_Global.station.MotionRow) + tSizeOfMotionRow,
						n:=			SIZEOF(gHMIMotionRows.gMotionRows)
						);
						
	retval := memcpy(	destAddr:=	ADR(S3_Global.station.MotionRowBtn) + tSizeOfMotionRowButtons,
						srcAddr:=	ADR(gHMIMotionRows.gMotionRowButtons),
						n:=			SIZEOF(gHMIMotionRows.gMotionRowButtons)
						);
END_IF

IF gHMIData.gStationSelected[4] THEN
	retval := memcpy(	destAddr:=	ADR(gHMIMotionRows.gMotionRows),
						srcAddr:=	ADR(S4_Global.station.MotionRow) + tSizeOfMotionRow,
						n:=			SIZEOF(gHMIMotionRows.gMotionRows)
						);
						
	retval := memcpy(	destAddr:=	ADR(S4_Global.station.MotionRowBtn) + tSizeOfMotionRowButtons,
						srcAddr:=	ADR(gHMIMotionRows.gMotionRowButtons),
						n:=			SIZEOF(gHMIMotionRows.gMotionRowButtons)
						);
END_IF

IF gHMIData.gStationSelected[5] THEN
	retval := memcpy(	destAddr:=	ADR(gHMIMotionRows.gMotionRows),
						srcAddr:=	ADR(S5_Global.station.MotionRow) + tSizeOfMotionRow,
						n:=			SIZEOF(gHMIMotionRows.gMotionRows)
						);
						
	retval := memcpy(	destAddr:=	ADR(S5_Global.station.MotionRowBtn) + tSizeOfMotionRowButtons,
						srcAddr:=	ADR(gHMIMotionRows.gMotionRowButtons),
						n:=			SIZEOF(gHMIMotionRows.gMotionRowButtons)
						);
END_IF

IF gHMIData.gStationSelected[6] THEN
	retval := memcpy(	destAddr:=	ADR(gHMIMotionRows.gMotionRows),
						srcAddr:=	ADR(S6_Global.station.MotionRow) + tSizeOfMotionRow,
						n:=			SIZEOF(gHMIMotionRows.gMotionRows)
						);
						
	retval := memcpy(	destAddr:=	ADR(S6_Global.station.MotionRowBtn) + tSizeOfMotionRowButtons,
						srcAddr:=	ADR(gHMIMotionRows.gMotionRowButtons),
						n:=			SIZEOF(gHMIMotionRows.gMotionRowButtons)
						);
END_IF
END_ACTION

ACTION actPageControl:
//imply TRIG call
btnNext(clk:=gHMIButtons.btnNextPage);
btnPrev(clk:=gHMIButtons.btnPrevPage);

//imply TRIG call
btnNextRow(clk:=gHMIButtons.btnPlus1Row); 
btnPrevRow(clk:=gHMIButtons.btnNeg1Row);

//next page
IF btnNext.Q THEN
	gHMIData.gActivePageNumber := gHMIData.gActivePageNumber + 1;
	
	//reset single offset
	tSingleRowOffsetFactor := 0;
END_IF

//previous page
IF btnPrev.Q THEN
	gHMIData.gActivePageNumber := gHMIData.gActivePageNumber - 1;
	
	//reset single offset
	tSingleRowOffsetFactor := 0;
END_IF

//apply limits
IF gHMIData.gActivePageNumber < 1 THEN
	gHMIData.gActivePageNumber := 1;
END_IF

//apply limits
IF gHMIData.gActivePageNumber > gHMIData.gMaxPageNumber THEN
	gHMIData.gActivePageNumber := gHMIData.gMaxPageNumber;
END_IF

//station 1 control
IF gHMIData.gStationSelected[1] THEN
	gHMIData.gMaxPageNumber := S1_Global.station.Data.NumberOfPages;
END_IF

//station 2 control
IF gHMIData.gStationSelected[2] THEN
	gHMIData.gMaxPageNumber := S2_Global.station.Data.NumberOfPages;
END_IF

//station 3 control
IF gHMIData.gStationSelected[3] THEN
	gHMIData.gMaxPageNumber := S3_Global.station.Data.NumberOfPages;
END_IF

//station 4 control
IF gHMIData.gStationSelected[4] THEN
	gHMIData.gMaxPageNumber := S4_Global.station.Data.NumberOfPages;
END_IF

//station 5 control
IF gHMIData.gStationSelected[5] THEN
	gHMIData.gMaxPageNumber := S5_Global.station.Data.NumberOfPages;
END_IF

//station 6 control
IF gHMIData.gStationSelected[6] THEN
	gHMIData.gMaxPageNumber := S6_Global.station.Data.NumberOfPages;
END_IF

//calc single row offset
//tSingleRowOffset
IF btnNextRow.Q THEN
tSingleRowOffsetFactor := tSingleRowOffsetFactor +1;
END_IF

IF btnPrevRow.Q THEN
tSingleRowOffsetFactor := tSingleRowOffsetFactor - 1;
END_IF

//single row cleanup
IF tSingleRowOffsetFactor >= 65535 THEN
	tSingleRowOffsetFactor := 0;
END_IF
END_ACTION

END_PROGRAM

// ---- HMI1/Logic/prgShowButtons.TcPOU
PROGRAM prgShowButtons
VAR
	tStationNumber: INT;
END_VAR

//hide all
actHideAll();

//if station is selected, then apply that stations mask to enable/hide functions
IF gHMIData.gStationSelected[1] THEN
	actHideAll_S_1();
END_IF

IF gHMIData.gStationSelected[2] THEN
	actHideAll_S_2();
END_IF

IF gHMIData.gStationSelected[3] THEN
	actHideAll_S_3();
END_IF

IF gHMIData.gStationSelected[4] THEN
	actHideAll_S_4();
END_IF

IF gHMIData.gStationSelected[5] THEN
	actHideAll_S_5();
END_IF

IF gHMIData.gStationSelected[6] THEN
	actHideAll_S_6();
END_IF

ACTION actHideAll:
//hide/show buttons on mode screen

//row 0
gHMIButtons.btnHides.btn00Hide := FALSE;
gHMIButtons.btnHides.btn01Hide := FALSE;
gHMIButtons.btnHides.btn02Hide := FALSE;
gHMIButtons.btnHides.btn03Hide := FALSE;
gHMIButtons.btnHides.btn04Hide := FALSE;
gHMIButtons.btnHides.btn05Hide := FALSE;
gHMIButtons.btnHides.btn06Hide := FALSE;
gHMIButtons.btnHides.btn07Hide := FALSE;
gHMIButtons.btnHides.btn08Hide := FALSE;
gHMIButtons.btnHides.btn09Hide := FALSE;

//row 1
gHMIButtons.btnHides.btn10Hide := FALSE;
gHMIButtons.btnHides.btn11Hide := FALSE;
gHMIButtons.btnHides.btn12Hide := FALSE;
gHMIButtons.btnHides.btn13Hide := FALSE;
gHMIButtons.btnHides.btn14Hide := FALSE;
gHMIButtons.btnHides.btn15Hide := FALSE;
gHMIButtons.btnHides.btn16Hide := FALSE;
gHMIButtons.btnHides.btn17Hide := FALSE;
gHMIButtons.btnHides.btn18Hide := FALSE;
gHMIButtons.btnHides.btn19Hide := FALSE;

//row 2
gHMIButtons.btnHides.btn20Hide := FALSE;
gHMIButtons.btnHides.btn21Hide := FALSE;
gHMIButtons.btnHides.btn22Hide := FALSE;
gHMIButtons.btnHides.btn23Hide := FALSE;
gHMIButtons.btnHides.btn24Hide := FALSE;
gHMIButtons.btnHides.btn25Hide := FALSE;
gHMIButtons.btnHides.btn26Hide := FALSE;
gHMIButtons.btnHides.btn27Hide := FALSE;
gHMIButtons.btnHides.btn28Hide := FALSE;
gHMIButtons.btnHides.btn29Hide := FALSE;

//row 3
gHMIButtons.btnHides.btn30Hide := FALSE;
gHMIButtons.btnHides.btn31Hide := FALSE;
gHMIButtons.btnHides.btn32Hide := FALSE;
gHMIButtons.btnHides.btn33Hide := FALSE;
gHMIButtons.btnHides.btn34Hide := FALSE;
gHMIButtons.btnHides.btn35Hide := FALSE;
gHMIButtons.btnHides.btn36Hide := FALSE;
gHMIButtons.btnHides.btn37Hide := FALSE;
gHMIButtons.btnHides.btn38Hide := FALSE;
gHMIButtons.btnHides.btn39Hide := FALSE;
END_ACTION

ACTION actHideAll_S_1:
//hide/show buttons on mode screen
tStationNumber:= 1;


//row 0
gHMIButtons.btnHides.btn00Hide := NOT System.gSetup.stationFunctions[tStationNumber].allowAutoCycle;
gHMIButtons.btnHides.btn01Hide := NOT System.gSetup.stationFunctions[tStationNumber].allowManualMode;
gHMIButtons.btnHides.btn02Hide := NOT System.gSetup.stationFunctions[tStationNumber].allowSemiAuto;
gHMIButtons.btnHides.btn03Hide := TRUE; //spare button
gHMIButtons.btnHides.btn04Hide := TRUE; //spare button
gHMIButtons.btnHides.btn05Hide := NOT System.gSetup.stationFunctions[tStationNumber].allowRemoteControl;
gHMIButtons.btnHides.btn06Hide := TRUE;
gHMIButtons.btnHides.btn07Hide := FALSE;
gHMIButtons.btnHides.btn08Hide := FALSE;
gHMIButtons.btnHides.btn09Hide := FALSE;

//row 1
gHMIButtons.btnHides.btn10Hide := NOT System.gSetup.stationFunctions[tStationNumber].allowContinuousCycle;
gHMIButtons.btnHides.btn11Hide := NOT System.gSetup.stationFunctions[tStationNumber].allowDryCycle;
gHMIButtons.btnHides.btn12Hide := NOT System.gSetup.stationFunctions[tStationNumber].allowSEOC;
gHMIButtons.btnHides.btn13Hide := NOT System.gSetup.stationFunctions[tStationNumber].allowSingleCycle;
gHMIButtons.btnHides.btn14Hide := TRUE; //spare button
gHMIButtons.btnHides.btn15Hide := NOT System.gSetup.stationFunctions[tStationNumber].allowSilenceHorn;
gHMIButtons.btnHides.btn16Hide := TRUE; //spare button
gHMIButtons.btnHides.btn17Hide := FALSE;
gHMIButtons.btnHides.btn18Hide := FALSE;
gHMIButtons.btnHides.btn19Hide := FALSE;

//row 2
gHMIButtons.btnHides.btn20Hide := NOT System.gSetup.stationFunctions[tStationNumber].allowGate1Req;
gHMIButtons.btnHides.btn21Hide := NOT System.gSetup.stationFunctions[tStationNumber].allowGate1Req;
gHMIButtons.btnHides.btn22Hide := NOT System.gSetup.stationFunctions[tStationNumber].allowLockAccessGates;
gHMIButtons.btnHides.btn23Hide := NOT System.gSetup.stationFunctions[tStationNumber].allowEnablePendent;
gHMIButtons.btnHides.btn24Hide := TRUE; //spare button
gHMIButtons.btnHides.btn25Hide := TRUE; //spare button
gHMIButtons.btnHides.btn26Hide := TRUE; //spare button
gHMIButtons.btnHides.btn27Hide := FALSE;
gHMIButtons.btnHides.btn28Hide := FALSE;
gHMIButtons.btnHides.btn29Hide := FALSE;

//row 3
gHMIButtons.btnHides.btn30Hide := FALSE;
gHMIButtons.btnHides.btn31Hide := FALSE;
gHMIButtons.btnHides.btn32Hide := FALSE;
gHMIButtons.btnHides.btn33Hide := FALSE;
gHMIButtons.btnHides.btn34Hide := FALSE;
gHMIButtons.btnHides.btn35Hide := FALSE;
gHMIButtons.btnHides.btn36Hide := FALSE;
gHMIButtons.btnHides.btn37Hide := FALSE;
gHMIButtons.btnHides.btn38Hide := FALSE;
gHMIButtons.btnHides.btn39Hide := FALSE;
END_ACTION

ACTION actHideAll_S_2:
//hide/show buttons on mode screen
tStationNumber:= 1;


//row 0
gHMIButtons.btnHides.btn00Hide := NOT System.gSetup.stationFunctions[tStationNumber].allowAutoCycle;
gHMIButtons.btnHides.btn01Hide := NOT System.gSetup.stationFunctions[tStationNumber].allowManualMode;
gHMIButtons.btnHides.btn02Hide := NOT System.gSetup.stationFunctions[tStationNumber].allowSemiAuto;
gHMIButtons.btnHides.btn03Hide := TRUE; //spare button
gHMIButtons.btnHides.btn04Hide := TRUE; //spare button
gHMIButtons.btnHides.btn05Hide := NOT System.gSetup.stationFunctions[tStationNumber].allowRemoteControl;
gHMIButtons.btnHides.btn06Hide := TRUE;
gHMIButtons.btnHides.btn07Hide := FALSE;
gHMIButtons.btnHides.btn08Hide := FALSE;
gHMIButtons.btnHides.btn09Hide := FALSE;

//row 1
gHMIButtons.btnHides.btn10Hide := NOT System.gSetup.stationFunctions[tStationNumber].allowContinuousCycle;
gHMIButtons.btnHides.btn11Hide := NOT System.gSetup.stationFunctions[tStationNumber].allowDryCycle;
gHMIButtons.btnHides.btn12Hide := NOT System.gSetup.stationFunctions[tStationNumber].allowSEOC;
gHMIButtons.btnHides.btn13Hide := NOT System.gSetup.stationFunctions[tStationNumber].allowSingleCycle;
gHMIButtons.btnHides.btn14Hide := TRUE; //spare button
gHMIButtons.btnHides.btn15Hide := NOT System.gSetup.stationFunctions[tStationNumber].allowSilenceHorn;
gHMIButtons.btnHides.btn16Hide := TRUE; //spare button
gHMIButtons.btnHides.btn17Hide := FALSE;
gHMIButtons.btnHides.btn18Hide := FALSE;
gHMIButtons.btnHides.btn19Hide := FALSE;

//row 2
gHMIButtons.btnHides.btn20Hide := NOT System.gSetup.stationFunctions[tStationNumber].allowGate1Req;
gHMIButtons.btnHides.btn21Hide := NOT System.gSetup.stationFunctions[tStationNumber].allowGate1Req;
gHMIButtons.btnHides.btn22Hide := NOT System.gSetup.stationFunctions[tStationNumber].allowLockAccessGates;
gHMIButtons.btnHides.btn23Hide := NOT System.gSetup.stationFunctions[tStationNumber].allowEnablePendent;
gHMIButtons.btnHides.btn24Hide := TRUE; //spare button
gHMIButtons.btnHides.btn25Hide := TRUE; //spare button
gHMIButtons.btnHides.btn26Hide := TRUE; //spare button
gHMIButtons.btnHides.btn27Hide := FALSE;
gHMIButtons.btnHides.btn28Hide := FALSE;
gHMIButtons.btnHides.btn29Hide := FALSE;

//row 3
gHMIButtons.btnHides.btn30Hide := FALSE;
gHMIButtons.btnHides.btn31Hide := FALSE;
gHMIButtons.btnHides.btn32Hide := FALSE;
gHMIButtons.btnHides.btn33Hide := FALSE;
gHMIButtons.btnHides.btn34Hide := FALSE;
gHMIButtons.btnHides.btn35Hide := FALSE;
gHMIButtons.btnHides.btn36Hide := FALSE;
gHMIButtons.btnHides.btn37Hide := FALSE;
gHMIButtons.btnHides.btn38Hide := FALSE;
gHMIButtons.btnHides.btn39Hide := FALSE;
END_ACTION

ACTION actHideAll_S_3:
//hide/show buttons on mode screen
tStationNumber:= 1;


//row 0
gHMIButtons.btnHides.btn00Hide := NOT System.gSetup.stationFunctions[tStationNumber].allowAutoCycle;
gHMIButtons.btnHides.btn01Hide := NOT System.gSetup.stationFunctions[tStationNumber].allowManualMode;
gHMIButtons.btnHides.btn02Hide := NOT System.gSetup.stationFunctions[tStationNumber].allowSemiAuto;
gHMIButtons.btnHides.btn03Hide := TRUE; //spare button
gHMIButtons.btnHides.btn04Hide := TRUE; //spare button
gHMIButtons.btnHides.btn05Hide := NOT System.gSetup.stationFunctions[tStationNumber].allowRemoteControl;
gHMIButtons.btnHides.btn06Hide := TRUE;
gHMIButtons.btnHides.btn07Hide := FALSE;
gHMIButtons.btnHides.btn08Hide := FALSE;
gHMIButtons.btnHides.btn09Hide := FALSE;

//row 1
gHMIButtons.btnHides.btn10Hide := NOT System.gSetup.stationFunctions[tStationNumber].allowContinuousCycle;
gHMIButtons.btnHides.btn11Hide := NOT System.gSetup.stationFunctions[tStationNumber].allowDryCycle;
gHMIButtons.btnHides.btn12Hide := NOT System.gSetup.stationFunctions[tStationNumber].allowSEOC;
gHMIButtons.btnHides.btn13Hide := NOT System.gSetup.stationFunctions[tStationNumber].allowSingleCycle;
gHMIButtons.btnHides.btn14Hide := TRUE; //spare button
gHMIButtons.btnHides.btn15Hide := NOT System.gSetup.stationFunctions[tStationNumber].allowSilenceHorn;
gHMIButtons.btnHides.btn16Hide := TRUE; //spare button
gHMIButtons.btnHides.btn17Hide := FALSE;
gHMIButtons.btnHides.btn18Hide := FALSE;
gHMIButtons.btnHides.btn19Hide := FALSE;

//row 2
gHMIButtons.btnHides.btn20Hide := NOT System.gSetup.stationFunctions[tStationNumber].allowGate1Req;
gHMIButtons.btnHides.btn21Hide := NOT System.gSetup.stationFunctions[tStationNumber].allowGate1Req;
gHMIButtons.btnHides.btn22Hide := NOT System.gSetup.stationFunctions[tStationNumber].allowLockAccessGates;
gHMIButtons.btnHides.btn23Hide := NOT System.gSetup.stationFunctions[tStationNumber].allowEnablePendent;
gHMIButtons.btnHides.btn24Hide := TRUE; //spare button
gHMIButtons.btnHides.btn25Hide := TRUE; //spare button
gHMIButtons.btnHides.btn26Hide := TRUE; //spare button
gHMIButtons.btnHides.btn27Hide := FALSE;
gHMIButtons.btnHides.btn28Hide := FALSE;
gHMIButtons.btnHides.btn29Hide := FALSE;

//row 3
gHMIButtons.btnHides.btn30Hide := FALSE;
gHMIButtons.btnHides.btn31Hide := FALSE;
gHMIButtons.btnHides.btn32Hide := FALSE;
gHMIButtons.btnHides.btn33Hide := FALSE;
gHMIButtons.btnHides.btn34Hide := FALSE;
gHMIButtons.btnHides.btn35Hide := FALSE;
gHMIButtons.btnHides.btn36Hide := FALSE;
gHMIButtons.btnHides.btn37Hide := FALSE;
gHMIButtons.btnHides.btn38Hide := FALSE;
gHMIButtons.btnHides.btn39Hide := FALSE;
END_ACTION

ACTION actHideAll_S_4:
//hide/show buttons on mode screen
tStationNumber:= 1;


//row 0
gHMIButtons.btnHides.btn00Hide := NOT System.gSetup.stationFunctions[tStationNumber].allowAutoCycle;
gHMIButtons.btnHides.btn01Hide := NOT System.gSetup.stationFunctions[tStationNumber].allowManualMode;
gHMIButtons.btnHides.btn02Hide := NOT System.gSetup.stationFunctions[tStationNumber].allowSemiAuto;
gHMIButtons.btnHides.btn03Hide := TRUE; //spare button
gHMIButtons.btnHides.btn04Hide := TRUE; //spare button
gHMIButtons.btnHides.btn05Hide := NOT System.gSetup.stationFunctions[tStationNumber].allowRemoteControl;
gHMIButtons.btnHides.btn06Hide := TRUE;
gHMIButtons.btnHides.btn07Hide := FALSE;
gHMIButtons.btnHides.btn08Hide := FALSE;
gHMIButtons.btnHides.btn09Hide := FALSE;

//row 1
gHMIButtons.btnHides.btn10Hide := NOT System.gSetup.stationFunctions[tStationNumber].allowContinuousCycle;
gHMIButtons.btnHides.btn11Hide := NOT System.gSetup.stationFunctions[tStationNumber].allowDryCycle;
gHMIButtons.btnHides.btn12Hide := NOT System.gSetup.stationFunctions[tStationNumber].allowSEOC;
gHMIButtons.btnHides.btn13Hide := NOT System.gSetup.stationFunctions[tStationNumber].allowSingleCycle;
gHMIButtons.btnHides.btn14Hide := TRUE; //spare button
gHMIButtons.btnHides.btn15Hide := NOT System.gSetup.stationFunctions[tStationNumber].allowSilenceHorn;
gHMIButtons.btnHides.btn16Hide := TRUE; //spare button
gHMIButtons.btnHides.btn17Hide := FALSE;
gHMIButtons.btnHides.btn18Hide := FALSE;
gHMIButtons.btnHides.btn19Hide := FALSE;

//row 2
gHMIButtons.btnHides.btn20Hide := NOT System.gSetup.stationFunctions[tStationNumber].allowGate1Req;
gHMIButtons.btnHides.btn21Hide := NOT System.gSetup.stationFunctions[tStationNumber].allowGate1Req;
gHMIButtons.btnHides.btn22Hide := NOT System.gSetup.stationFunctions[tStationNumber].allowLockAccessGates;
gHMIButtons.btnHides.btn23Hide := NOT System.gSetup.stationFunctions[tStationNumber].allowEnablePendent;
gHMIButtons.btnHides.btn24Hide := TRUE; //spare button
gHMIButtons.btnHides.btn25Hide := TRUE; //spare button
gHMIButtons.btnHides.btn26Hide := TRUE; //spare button
gHMIButtons.btnHides.btn27Hide := FALSE;
gHMIButtons.btnHides.btn28Hide := FALSE;
gHMIButtons.btnHides.btn29Hide := FALSE;

//row 3
gHMIButtons.btnHides.btn30Hide := FALSE;
gHMIButtons.btnHides.btn31Hide := FALSE;
gHMIButtons.btnHides.btn32Hide := FALSE;
gHMIButtons.btnHides.btn33Hide := FALSE;
gHMIButtons.btnHides.btn34Hide := FALSE;
gHMIButtons.btnHides.btn35Hide := FALSE;
gHMIButtons.btnHides.btn36Hide := FALSE;
gHMIButtons.btnHides.btn37Hide := FALSE;
gHMIButtons.btnHides.btn38Hide := FALSE;
gHMIButtons.btnHides.btn39Hide := FALSE;
END_ACTION

ACTION actHideAll_S_5:
//hide/show buttons on mode screen
tStationNumber:= 1;


//row 0
gHMIButtons.btnHides.btn00Hide := NOT System.gSetup.stationFunctions[tStationNumber].allowAutoCycle;
gHMIButtons.btnHides.btn01Hide := NOT System.gSetup.stationFunctions[tStationNumber].allowManualMode;
gHMIButtons.btnHides.btn02Hide := NOT System.gSetup.stationFunctions[tStationNumber].allowSemiAuto;
gHMIButtons.btnHides.btn03Hide := TRUE; //spare button
gHMIButtons.btnHides.btn04Hide := TRUE; //spare button
gHMIButtons.btnHides.btn05Hide := NOT System.gSetup.stationFunctions[tStationNumber].allowRemoteControl;
gHMIButtons.btnHides.btn06Hide := TRUE;
gHMIButtons.btnHides.btn07Hide := FALSE;
gHMIButtons.btnHides.btn08Hide := FALSE;
gHMIButtons.btnHides.btn09Hide := FALSE;

//row 1
gHMIButtons.btnHides.btn10Hide := NOT System.gSetup.stationFunctions[tStationNumber].allowContinuousCycle;
gHMIButtons.btnHides.btn11Hide := NOT System.gSetup.stationFunctions[tStationNumber].allowDryCycle;
gHMIButtons.btnHides.btn12Hide := NOT System.gSetup.stationFunctions[tStationNumber].allowSEOC;
gHMIButtons.btnHides.btn13Hide := NOT System.gSetup.stationFunctions[tStationNumber].allowSingleCycle;
gHMIButtons.btnHides.btn14Hide := TRUE; //spare button
gHMIButtons.btnHides.btn15Hide := NOT System.gSetup.stationFunctions[tStationNumber].allowSilenceHorn;
gHMIButtons.btnHides.btn16Hide := TRUE; //spare button
gHMIButtons.btnHides.btn17Hide := FALSE;
gHMIButtons.btnHides.btn18Hide := FALSE;
gHMIButtons.btnHides.btn19Hide := FALSE;

//row 2
gHMIButtons.btnHides.btn20Hide := NOT System.gSetup.stationFunctions[tStationNumber].allowGate1Req;
gHMIButtons.btnHides.btn21Hide := NOT System.gSetup.stationFunctions[tStationNumber].allowGate1Req;
gHMIButtons.btnHides.btn22Hide := NOT System.gSetup.stationFunctions[tStationNumber].allowLockAccessGates;
gHMIButtons.btnHides.btn23Hide := NOT System.gSetup.stationFunctions[tStationNumber].allowEnablePendent;
gHMIButtons.btnHides.btn24Hide := TRUE; //spare button
gHMIButtons.btnHides.btn25Hide := TRUE; //spare button
gHMIButtons.btnHides.btn26Hide := TRUE; //spare button
gHMIButtons.btnHides.btn27Hide := FALSE;
gHMIButtons.btnHides.btn28Hide := FALSE;
gHMIButtons.btnHides.btn29Hide := FALSE;

//row 3
gHMIButtons.btnHides.btn30Hide := FALSE;
gHMIButtons.btnHides.btn31Hide := FALSE;
gHMIButtons.btnHides.btn32Hide := FALSE;
gHMIButtons.btnHides.btn33Hide := FALSE;
gHMIButtons.btnHides.btn34Hide := FALSE;
gHMIButtons.btnHides.btn35Hide := FALSE;
gHMIButtons.btnHides.btn36Hide := FALSE;
gHMIButtons.btnHides.btn37Hide := FALSE;
gHMIButtons.btnHides.btn38Hide := FALSE;
gHMIButtons.btnHides.btn39Hide := FALSE;
END_ACTION

ACTION actHideAll_S_6:
//hide/show buttons on mode screen
tStationNumber:= 1;


//row 0
gHMIButtons.btnHides.btn00Hide := NOT System.gSetup.stationFunctions[tStationNumber].allowAutoCycle;
gHMIButtons.btnHides.btn01Hide := NOT System.gSetup.stationFunctions[tStationNumber].allowManualMode;
gHMIButtons.btnHides.btn02Hide := NOT System.gSetup.stationFunctions[tStationNumber].allowSemiAuto;
gHMIButtons.btnHides.btn03Hide := TRUE; //spare button
gHMIButtons.btnHides.btn04Hide := TRUE; //spare button
gHMIButtons.btnHides.btn05Hide := NOT System.gSetup.stationFunctions[tStationNumber].allowRemoteControl;
gHMIButtons.btnHides.btn06Hide := TRUE;
gHMIButtons.btnHides.btn07Hide := FALSE;
gHMIButtons.btnHides.btn08Hide := FALSE;
gHMIButtons.btnHides.btn09Hide := FALSE;

//row 1
gHMIButtons.btnHides.btn10Hide := NOT System.gSetup.stationFunctions[tStationNumber].allowContinuousCycle;
gHMIButtons.btnHides.btn11Hide := NOT System.gSetup.stationFunctions[tStationNumber].allowDryCycle;
gHMIButtons.btnHides.btn12Hide := NOT System.gSetup.stationFunctions[tStationNumber].allowSEOC;
gHMIButtons.btnHides.btn13Hide := NOT System.gSetup.stationFunctions[tStationNumber].allowSingleCycle;
gHMIButtons.btnHides.btn14Hide := TRUE; //spare button
gHMIButtons.btnHides.btn15Hide := NOT System.gSetup.stationFunctions[tStationNumber].allowSilenceHorn;
gHMIButtons.btnHides.btn16Hide := TRUE; //spare button
gHMIButtons.btnHides.btn17Hide := FALSE;
gHMIButtons.btnHides.btn18Hide := FALSE;
gHMIButtons.btnHides.btn19Hide := FALSE;

//row 2
gHMIButtons.btnHides.btn20Hide := NOT System.gSetup.stationFunctions[tStationNumber].allowGate1Req;
gHMIButtons.btnHides.btn21Hide := NOT System.gSetup.stationFunctions[tStationNumber].allowGate1Req;
gHMIButtons.btnHides.btn22Hide := NOT System.gSetup.stationFunctions[tStationNumber].allowLockAccessGates;
gHMIButtons.btnHides.btn23Hide := NOT System.gSetup.stationFunctions[tStationNumber].allowEnablePendent;
gHMIButtons.btnHides.btn24Hide := TRUE; //spare button
gHMIButtons.btnHides.btn25Hide := TRUE; //spare button
gHMIButtons.btnHides.btn26Hide := TRUE; //spare button
gHMIButtons.btnHides.btn27Hide := FALSE;
gHMIButtons.btnHides.btn28Hide := FALSE;
gHMIButtons.btnHides.btn29Hide := FALSE;

//row 3
gHMIButtons.btnHides.btn30Hide := FALSE;
gHMIButtons.btnHides.btn31Hide := FALSE;
gHMIButtons.btnHides.btn32Hide := FALSE;
gHMIButtons.btnHides.btn33Hide := FALSE;
gHMIButtons.btnHides.btn34Hide := FALSE;
gHMIButtons.btnHides.btn35Hide := FALSE;
gHMIButtons.btnHides.btn36Hide := FALSE;
gHMIButtons.btnHides.btn37Hide := FALSE;
gHMIButtons.btnHides.btn38Hide := FALSE;
gHMIButtons.btnHides.btn39Hide := FALSE;
END_ACTION

END_PROGRAM

// ---- HMI1/Logic/prgHMIUnits.TcPOU
PROGRAM prgHMIUnits
VAR
	tTrueUnitIndex: UINT;
	tSizeOfUnitRow: UINT;
	tSizeOfUnitRowButtons: UINT;
	tStationNumberIndexUnit: UINT;
	tScreenElementsPerPageUnit: UINT;
	tNumElementsPerScreen: UINT;
	retval: UDINT;
	nextPage: R_TRIG;
	PrevPage: R_TRIG;
END_VAR

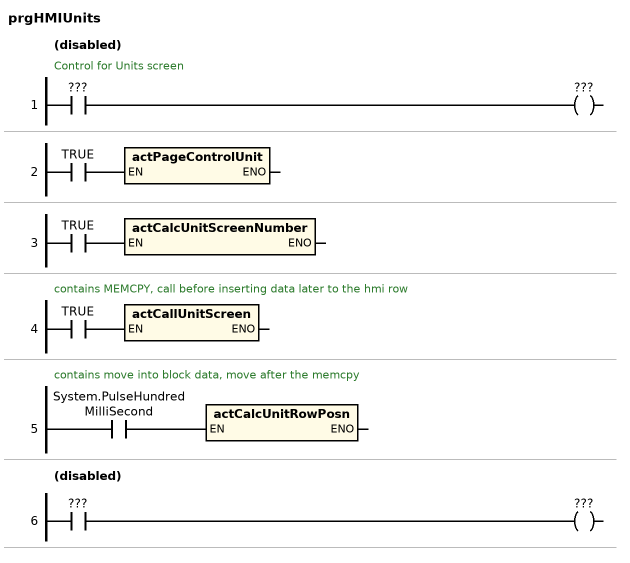
// NETWORK 1 (disabled)
// Control for Units screen
// ??? := ???;

// NETWORK 2
actPageControlUnit();

// NETWORK 3
actCalcUnitScreenNumber();

// NETWORK 4
// contains MEMCPY, call before inserting data later to the hmi row
actCallUnitScreen();

// NETWORK 5
// contains move into block data, move after the memcpy
IF System.PulseHundredMilliSecond THEN actCalcUnitRowPosn(); END_IF

// NETWORK 6 (disabled)
// ??? := ???;

ACTION actCalcUnitRowPosn:
//calculate station index for pages
tTrueUnitIndex :=	tStationNumberIndexUnit +
					(tScreenElementsPerPageUnit * gHMIUnits.gUnitActivePageNumber) -  tScreenElementsPerPageUnit;
					
//calculate offset for row x
gHMIUnits.gUnitRowElementOffset[1] :=	tTrueUnitIndex + 
										(gHMIDataConst.gNumberElementsPerRow * 1) - gHMIDataConst.gNumberElementsPerRow;

gHMIUnits.gUnitRowElementOffset[2] :=	tTrueUnitIndex + 
										(gHMIDataConst.gNumberElementsPerRow * 2) - gHMIDataConst.gNumberElementsPerRow;

gHMIUnits.gUnitRowElementOffset[3] :=	tTrueUnitIndex + 
										(gHMIDataConst.gNumberElementsPerRow * 3) - gHMIDataConst.gNumberElementsPerRow;

gHMIUnits.gUnitRowElementOffset[4] :=	tTrueUnitIndex + 
										(gHMIDataConst.gNumberElementsPerRow * 4) - gHMIDataConst.gNumberElementsPerRow;

gHMIUnits.gUnitRowElementOffset[5] :=	tTrueUnitIndex + 
										(gHMIDataConst.gNumberElementsPerRow * 5) - gHMIDataConst.gNumberElementsPerRow;

gHMIUnits.gUnitRowElementOffset[6] :=	tTrueUnitIndex + 
										(gHMIDataConst.gNumberElementsPerRow * 6) - gHMIDataConst.gNumberElementsPerRow;
				
//move to global to be picked up by each row					
gHMIUnits.gUnitRows.gMotionRow1.IndexLocation := gHMIUnits.gUnitRowElementOffset[1];
gHMIUnits.gUnitRows.gMotionRow2.IndexLocation := gHMIUnits.gUnitRowElementOffset[2];
gHMIUnits.gUnitRows.gMotionRow3.IndexLocation := gHMIUnits.gUnitRowElementOffset[3];
gHMIUnits.gUnitRows.gMotionRow4.IndexLocation := gHMIUnits.gUnitRowElementOffset[4];
gHMIUnits.gUnitRows.gMotionRow5.IndexLocation := gHMIUnits.gUnitRowElementOffset[5];
gHMIUnits.gUnitRows.gMotionRow6.IndexLocation := gHMIUnits.gUnitRowElementOffset[6];
END_ACTION

ACTION actCalcUnitScreenNumber:
//create number for station
tStationNumberIndexUnit	:= 1 * 10000; //declare math for now


//calculate number of elements per screen
tNumElementsPerScreen	:= gHMIDataConst.gNumberRowsPerPage * gHMIDataConst.gNumberElementsPerRow;

//calculate screen per page index
tScreenElementsPerPageUnit := tNumElementsPerScreen * 1; //declare math for future use
END_ACTION

ACTION actCallUnitScreen:
//calculate byte offset - motions
tSizeOfUnitRow := gHMIData.gActivePageNumber * SIZEOF(gHMIUnits.gUnitRows); //for pointer use
tSizeOfUnitRow := tSizeOfUnitRow - SIZEOF(gHMIUnits.gUnitRows);

//calculate byte offset - buttons
tSizeOfUnitRowButtons := gHMIData.gActivePageNumber * SIZEOF(gHMIUnits.gUnitButtons);
tSizeOfUnitRowButtons := tSizeOfUnitRowButtons - SIZEOF(gHMIUnits.gUnitButtons);

//move data based on station and page number
//Move feedback indicator data
//Move Button BOOL state back adr(S1_Global.MotionRow)
MEMCPY(	destAddr	:= ADR(gHMIUnits.gUnitRows),
		srcAddr		:= ADR(Mc_Global.UnitRow) + tSizeOfUnitRow,
		n			:= SIZEOF(gHMIData.gLangRows)
		);

MEMCPY(	destAddr	:= ADR(Mc_Global.UnitRowBtn) + tSizeOfUnitRowButtons,
		srcAddr		:= ADR(gHMIUnits.gUnitButtons),
		n			:= SIZEOF(gHMIUnits.gUnitButtons)
		);
END_ACTION

ACTION actPageControlUnit:
//next page
nextPage(CLK	:= gHMIButtons.btnNextPage);
IF nextPage.Q THEN
	gHMIUnits.gUnitActivePageNumber	:=	gHMIUnits.gUnitActivePageNumber + 1;
END_IF

//previous page
PrevPage(CLK	:= gHMIButtons.btnPrevPage);
IF PrevPage.Q THEN
	gHMIUnits.gUnitActivePageNumber := gHMIUnits.gUnitActivePageNumber - 1;
END_IF



//apply limits
IF gHMIUnits.gUnitActivePageNumber < 1 THEN
	gHMIUnits.gUnitActivePageNumber := 1;
END_IF
	
IF gHMIUnits.gUnitActivePageNumber > gHMIUnits.gUnitMaxPageNumber THEN
	gHMIUnits.gUnitActivePageNumber := 1;
END_IF

gHMIUnits.gUnitMaxPageNumber := Mc_Global.Data.NumberOfPages;
END_ACTION

END_PROGRAM

// ---- HMI1/Logic/prgHMIstations.TcPOU
PROGRAM prgHMIstations
VAR
		tAllStations: BOOL;
	tUsestaions: BOOL;
	btnselectalltrig: R_TRIG;
	btnselall: F_TRIG;
	btnselS1: R_TRIG;
	btnselS2: R_TRIG;
	btnselS3: R_TRIG;
	btnselS4: R_TRIG;
	btnselS5: R_TRIG;
	btnselS6: R_TRIG;

	tPulseStationSelect: BOOL;
	timDelayPulseSelect: TON;
	timPulseStationSelect:TP;
	
END_VAR

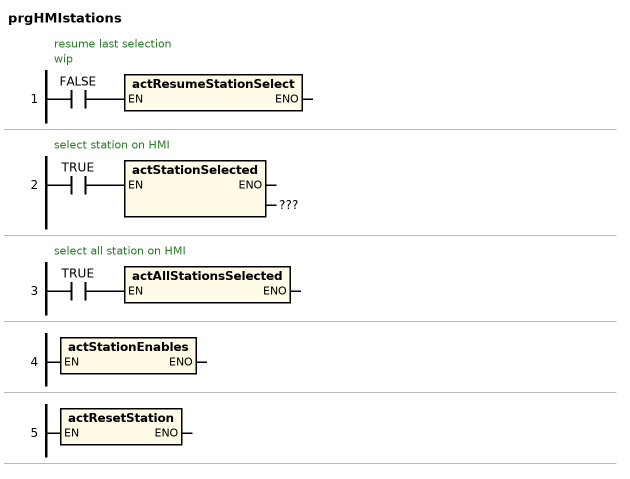
// NETWORK 1
// resume last selection
// wip
IF FALSE THEN actResumeStationSelect(); END_IF

// NETWORK 2
// select station on HMI
actStationSelected();

// NETWORK 3
// select all station on HMI
actAllStationsSelected();

// NETWORK 4
actStationEnables();

// NETWORK 5
actResetStation();

ACTION actAllStationsSelected:
//all station feedback
IF	gHMIData.gStationSelected[1]	AND	
	gHMIData.gStationSelected[2]	AND 
	gHMIData.gStationSelected[3]	AND
	gHMIData.gStationSelected[4]	AND
	gHMIData.gStationSelected[5]	AND
	gHMIData.gStationSelected[6]	
	THEN
		gHMIButtons.btnAllStationsSelected := TRUE;
	ELSE
		gHMIButtons.btnAllStationsSelected := FALSE;
END_IF

//select all stations
btnselectalltrig(CLK:= gHMIButtons.btnSelectAll);
IF btnselectalltrig.Q AND NOT gHMIButtons.btnAllStationsSelected THEN
	gHMIData.gStationSelected[1] := TRUE;
	gHMIData.gStationSelected[2] := TRUE;
	gHMIData.gStationSelected[3] := TRUE;
	gHMIData.gStationSelected[4] := TRUE;
	gHMIData.gStationSelected[5] := TRUE;
	gHMIData.gStationSelected[6] := TRUE;	
END_IF
END_ACTION

ACTION actResetStation:
//if no station is selected, then select station 1
//all station feedback
IF	NOT gHMIData.gStationSelected[1]	AND	
	NOT gHMIData.gStationSelected[2]	AND 
	NOT gHMIData.gStationSelected[3]	AND
	NOT gHMIData.gStationSelected[4]	AND
	NOT gHMIData.gStationSelected[5]	AND
	NOT gHMIData.gStationSelected[6]	
	THEN
		tPulseStationSelect := TRUE;
	ELSE
		tPulseStationSelect := FALSE;
END_IF

//timer delay
timDelayPulseSelect(IN:= tPulseStationSelect, PT:=T#10S);
timPulseStationSelect(IN:=timDelayPulseSelect.Q, PT:=T#1S);

IF timPulseStationSelect.Q THEN
	gHMIData.gActiveStationNumber := 1;
	gHMIData.gStationSelected[1] := TRUE;
END_IF
END_ACTION

ACTION actResumeStationSelect:
//all station feedback
//on select all button falling
btnselall(CLK:= gHMIButtons.btnSelectAll);
IF 	btnselall.Q 					AND
	gHMIData.gStationSelected[1]	AND 
	gHMIData.gStationSelected[2]	AND 
	gHMIData.gStationSelected[3]	AND 
	gHMIData.gStationSelected[4]	AND 
	gHMIData.gStationSelected[5]	AND 
	gHMIData.gStationSelected[6]	 
	THEN

	//clear out selected	
	IF gHMIData.gActiveStationNumber > 1 THEN
		gHMIData.gStationSelected[1] := FALSE;
		gHMIData.gStationSelected[2] := FALSE;
		gHMIData.gStationSelected[3] := FALSE;
		gHMIData.gStationSelected[4] := FALSE;
		gHMIData.gStationSelected[5] := FALSE;
		gHMIData.gStationSelected[6] := FALSE;
	END_IF
	
	//select correct station
	CASE gHMIData.gActiveStationNumber OF
		1:
		gHMIData.gStationSelected[1] := TRUE;
		2:
		gHMIData.gStationSelected[2] := TRUE;
		3:
		gHMIData.gStationSelected[3] := TRUE;
		4:
		gHMIData.gStationSelected[4] := TRUE;
		5:
		gHMIData.gStationSelected[5] := TRUE;
		6:
		gHMIData.gStationSelected[6] := TRUE;
	END_CASE
END_IF
END_ACTION

ACTION actStationEnables:
//disable all stations and let station calls enable on a per-scan basis
gHMIData.gStationEnabled[1]:= System.gSetup.stationEnable[1];
gHMIData.gStationEnabled[2]:= System.gSetup.stationEnable[2];
gHMIData.gStationEnabled[3]:= System.gSetup.stationEnable[3];
gHMIData.gStationEnabled[4]:= System.gSetup.stationEnable[4];
gHMIData.gStationEnabled[5]:= System.gSetup.stationEnable[5];
gHMIData.gStationEnabled[6]:= System.gSetup.stationEnable[6];
END_ACTION

ACTION actStationSelected:
//select station on HMI
//theme:czWR1tA8oB0

btnselS1(clk:=gHMIButtons.btnSelectStation1);
btnselS2(clk:=gHMIButtons.btnSelectStation2);
btnselS3(clk:=gHMIButtons.btnSelectStation3);
btnselS4(clk:=gHMIButtons.btnSelectStation4);
btnselS5(clk:=gHMIButtons.btnSelectStation5);
btnselS6(clk:=gHMIButtons.btnSelectStation6);


//if any button pressed, clear down station memory and prepare for new station selected data
IF	btnselS1.Q OR
	btnselS2.Q OR
	btnselS3.Q OR
	btnselS4.Q OR
	btnselS5.Q OR
	btnselS6.Q
	THEN
		MEMSET(	destAddr:= ADR(gHMIData.gStationSelected),
				fillByte:= 16#0,
				n		:= SIZEOF(gHMIData.gStationSelected)
				);
		gHMIData.gActivePageNumber := 1;
END_IF

//move in correct data next in scan
IF btnselS1.Q THEN
	gHMIData.gActiveStationNumber := 1;
	gHMIData.gStationSelected[1] := TRUE;
END_IF

IF btnselS2.Q THEN
	gHMIData.gActiveStationNumber := 2;
	gHMIData.gStationSelected[2] := TRUE;
END_IF

IF btnselS3.Q THEN
	gHMIData.gActiveStationNumber := 3;
	gHMIData.gStationSelected[3] := TRUE;
END_IF

IF btnselS4.Q THEN
	gHMIData.gActiveStationNumber := 4;
	gHMIData.gStationSelected[4] := TRUE;
END_IF

IF btnselS5.Q THEN
	gHMIData.gActiveStationNumber := 5;
	gHMIData.gStationSelected[5] := TRUE;
END_IF

IF btnselS6.Q THEN
	gHMIData.gActiveStationNumber := 6;
	gHMIData.gStationSelected[6] := TRUE;
END_IF
END_ACTION

END_PROGRAM

// ---- HMI1/Logic/prgReadTextList.TcPOU
PROGRAM prgReadTextList
VAR_INPUT
END_VAR
VAR_OUTPUT
END_VAR
VAR
	starttt: BOOL;
	readMC_Alarms: FB_ReadTextList;
	readMC_Prompts: FB_ReadTextList;
	readMC_Warnings: FB_ReadTextList;
	resett: BOOL;
	readS1_Alarms: FB_ReadTextList;
	readS1_Prompts: FB_ReadTextList;
	readS1_Warnings: FB_ReadTextList;
	
	readS2_Alarms: FB_ReadTextList;
	readS2_Prompts: FB_ReadTextList;
	readS2_Warnings: FB_ReadTextList;
	
	readS3_Alarms: FB_ReadTextList;
	readS3_Prompts: FB_ReadTextList;
	readS3_Warnings: FB_ReadTextList;
	
	readS4_Alarms: FB_ReadTextList;
	readS4_Prompts: FB_ReadTextList;
	readS4_Warnings: FB_ReadTextList;
	
	readS5_Alarms: FB_ReadTextList;
	readS5_Prompts: FB_ReadTextList;
	readS5_Warnings: FB_ReadTextList;
	
	readS6_Alarms: FB_ReadTextList;
	readS6_Prompts: FB_ReadTextList;
	readS6_Warnings: FB_ReadTextList;
	
	

	
END_VAR
VAR // added by the converter: edge detectors and wires of the graphical bodies
    _rt1, _rt2, _rt3, _rt4 : R_TRIG;
END_VAR

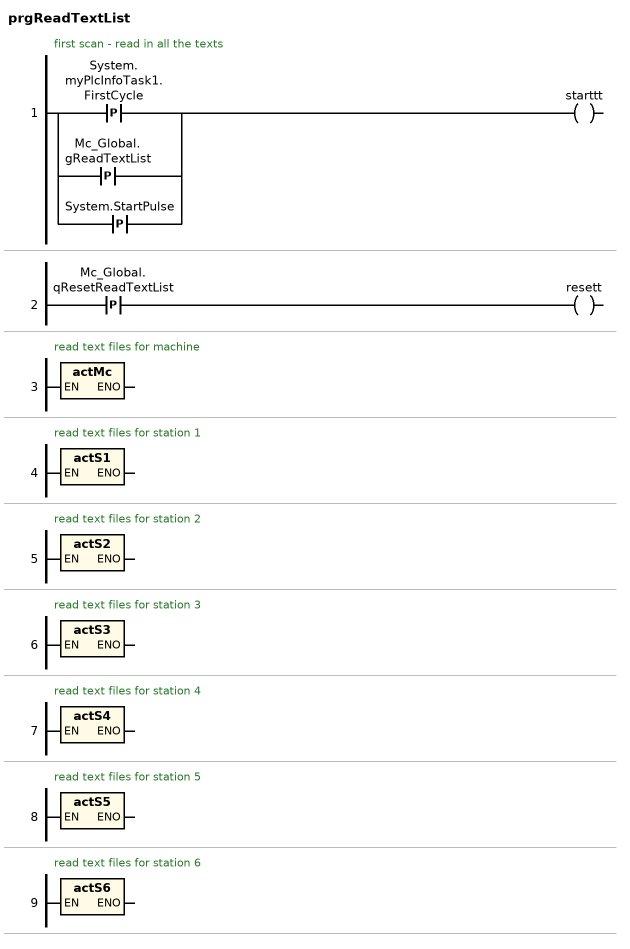
// NETWORK 1
// first scan - read in all the texts
_rt1(CLK := System.myPlcInfoTask1.FirstCycle);
_rt2(CLK := Mc_Global.gReadTextList);
_rt3(CLK := System.StartPulse);
starttt := _rt1.Q OR _rt2.Q OR _rt3.Q;

// NETWORK 2
_rt4(CLK := Mc_Global.qResetReadTextList);
resett := _rt4.Q;

// NETWORK 3
// read text files for machine
actMc();

// NETWORK 4
// read text files for station 1
actS1();

// NETWORK 5
// read text files for station 2
actS2();

// NETWORK 6
// read text files for station 3
actS3();

// NETWORK 7
// read text files for station 4
actS4();

// NETWORK 8
// read text files for station 5
actS5();

// NETWORK 9
// read text files for station 6
actS6();

ACTION actMc:
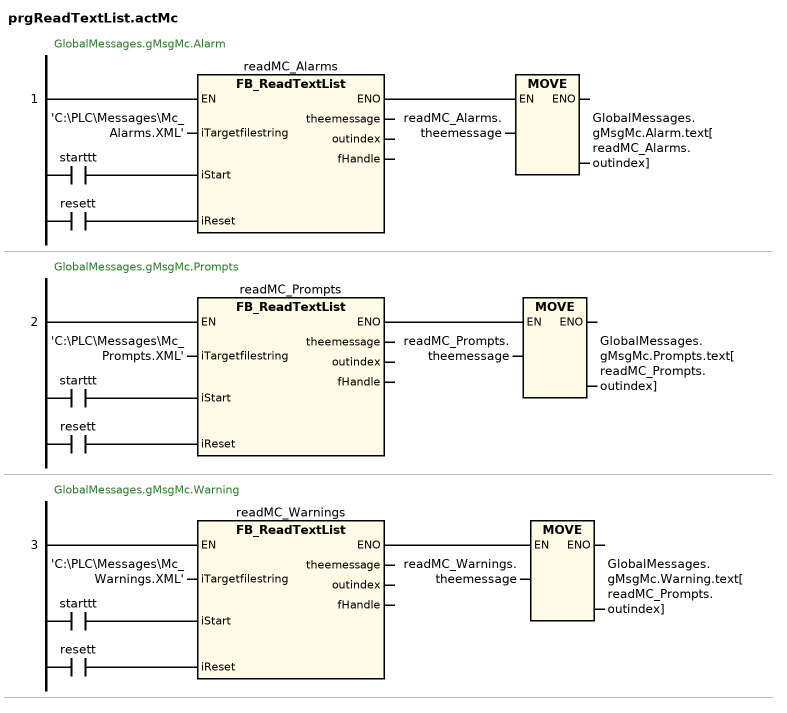
// NETWORK 1
// GlobalMessages.gMsgMc.Alarm
readMC_Alarms(iTargetfilestring := 'C:\PLC\Messages\Mc_Alarms.XML', iStart := starttt, iReset := resett); // FB_ReadTextList
GlobalMessages.gMsgMc.Alarm.text[readMC_Alarms.outindex] := readMC_Alarms.theemessage;

// NETWORK 2
// GlobalMessages.gMsgMc.Prompts
readMC_Prompts(iTargetfilestring := 'C:\PLC\Messages\Mc_Prompts.XML', iStart := starttt, iReset := resett); // FB_ReadTextList
GlobalMessages.gMsgMc.Prompts.text[readMC_Prompts.outindex] := readMC_Prompts.theemessage;

// NETWORK 3
// GlobalMessages.gMsgMc.Warning
readMC_Warnings(iTargetfilestring := 'C:\PLC\Messages\Mc_Warnings.XML', iStart := starttt, iReset := resett); // FB_ReadTextList
GlobalMessages.gMsgMc.Warning.text[readMC_Prompts.outindex] := readMC_Warnings.theemessage;
END_ACTION

ACTION actS1:
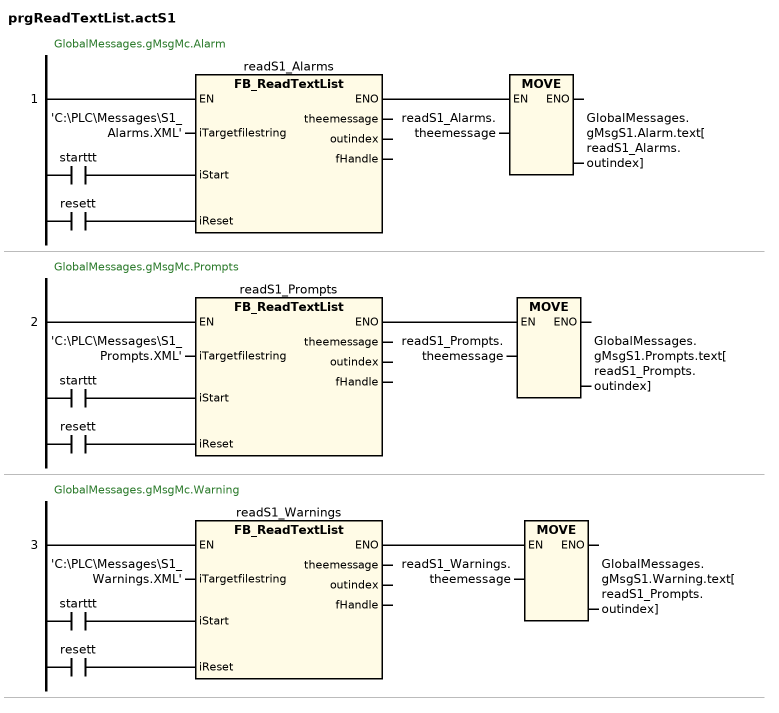
// NETWORK 1
// GlobalMessages.gMsgMc.Alarm
readS1_Alarms(iTargetfilestring := 'C:\PLC\Messages\S1_Alarms.XML', iStart := starttt, iReset := resett); // FB_ReadTextList
GlobalMessages.gMsgS1.Alarm.text[readS1_Alarms.outindex] := readS1_Alarms.theemessage;

// NETWORK 2
// GlobalMessages.gMsgMc.Prompts
readS1_Prompts(iTargetfilestring := 'C:\PLC\Messages\S1_Prompts.XML', iStart := starttt, iReset := resett); // FB_ReadTextList
GlobalMessages.gMsgS1.Prompts.text[readS1_Prompts.outindex] := readS1_Prompts.theemessage;

// NETWORK 3
// GlobalMessages.gMsgMc.Warning
readS1_Warnings(iTargetfilestring := 'C:\PLC\Messages\S1_Warnings.XML', iStart := starttt, iReset := resett); // FB_ReadTextList
GlobalMessages.gMsgS1.Warning.text[readS1_Prompts.outindex] := readS1_Warnings.theemessage;
END_ACTION

ACTION actS2:
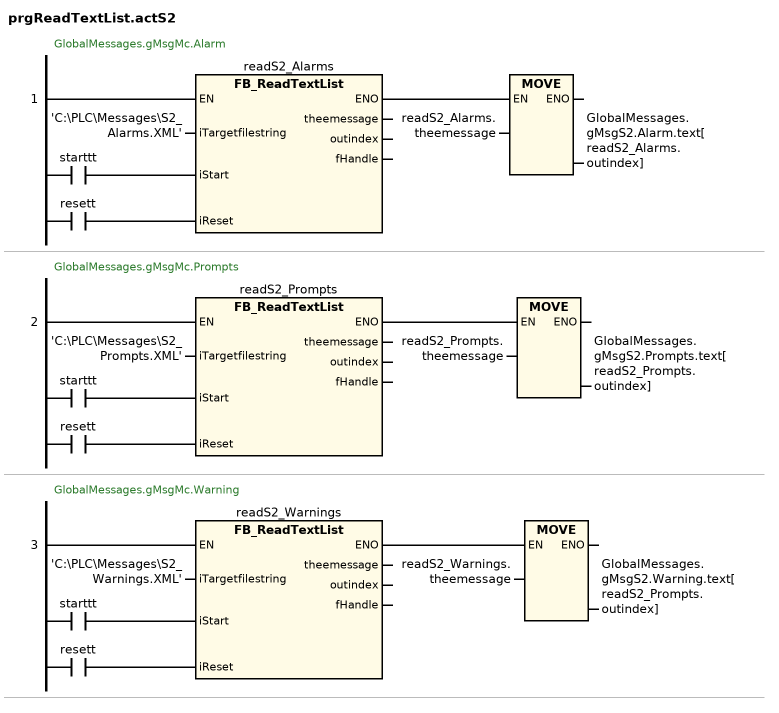
// NETWORK 1
// GlobalMessages.gMsgMc.Alarm
readS2_Alarms(iTargetfilestring := 'C:\PLC\Messages\S2_Alarms.XML', iStart := starttt, iReset := resett); // FB_ReadTextList
GlobalMessages.gMsgS2.Alarm.text[readS2_Alarms.outindex] := readS2_Alarms.theemessage;

// NETWORK 2
// GlobalMessages.gMsgMc.Prompts
readS2_Prompts(iTargetfilestring := 'C:\PLC\Messages\S2_Prompts.XML', iStart := starttt, iReset := resett); // FB_ReadTextList
GlobalMessages.gMsgS2.Prompts.text[readS2_Prompts.outindex] := readS2_Prompts.theemessage;

// NETWORK 3
// GlobalMessages.gMsgMc.Warning
readS2_Warnings(iTargetfilestring := 'C:\PLC\Messages\S2_Warnings.XML', iStart := starttt, iReset := resett); // FB_ReadTextList
GlobalMessages.gMsgS2.Warning.text[readS2_Prompts.outindex] := readS2_Warnings.theemessage;
END_ACTION

ACTION actS3:
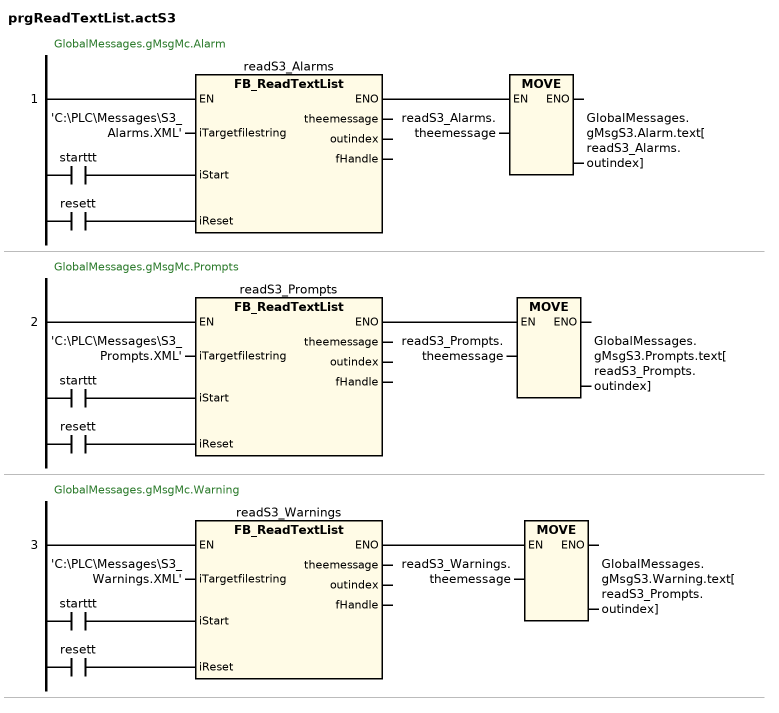
// NETWORK 1
// GlobalMessages.gMsgMc.Alarm
readS3_Alarms(iTargetfilestring := 'C:\PLC\Messages\S3_Alarms.XML', iStart := starttt, iReset := resett); // FB_ReadTextList
GlobalMessages.gMsgS3.Alarm.text[readS3_Alarms.outindex] := readS3_Alarms.theemessage;

// NETWORK 2
// GlobalMessages.gMsgMc.Prompts
readS3_Prompts(iTargetfilestring := 'C:\PLC\Messages\S3_Prompts.XML', iStart := starttt, iReset := resett); // FB_ReadTextList
GlobalMessages.gMsgS3.Prompts.text[readS3_Prompts.outindex] := readS3_Prompts.theemessage;

// NETWORK 3
// GlobalMessages.gMsgMc.Warning
readS3_Warnings(iTargetfilestring := 'C:\PLC\Messages\S3_Warnings.XML', iStart := starttt, iReset := resett); // FB_ReadTextList
GlobalMessages.gMsgS3.Warning.text[readS3_Prompts.outindex] := readS3_Warnings.theemessage;
END_ACTION

ACTION actS4:
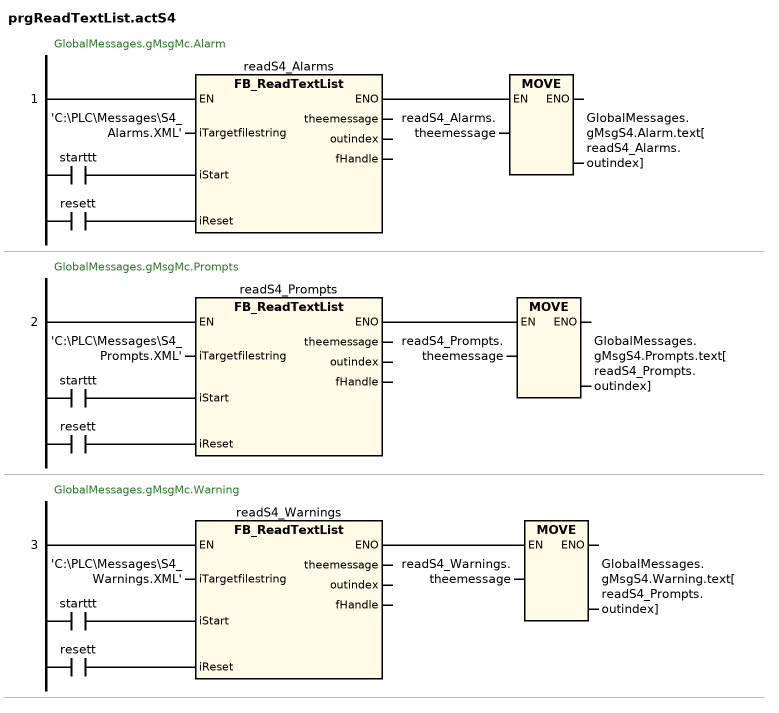
// NETWORK 1
// GlobalMessages.gMsgMc.Alarm
readS4_Alarms(iTargetfilestring := 'C:\PLC\Messages\S4_Alarms.XML', iStart := starttt, iReset := resett); // FB_ReadTextList
GlobalMessages.gMsgS4.Alarm.text[readS4_Alarms.outindex] := readS4_Alarms.theemessage;

// NETWORK 2
// GlobalMessages.gMsgMc.Prompts
readS4_Prompts(iTargetfilestring := 'C:\PLC\Messages\S4_Prompts.XML', iStart := starttt, iReset := resett); // FB_ReadTextList
GlobalMessages.gMsgS4.Prompts.text[readS4_Prompts.outindex] := readS4_Prompts.theemessage;

// NETWORK 3
// GlobalMessages.gMsgMc.Warning
readS4_Warnings(iTargetfilestring := 'C:\PLC\Messages\S4_Warnings.XML', iStart := starttt, iReset := resett); // FB_ReadTextList
GlobalMessages.gMsgS4.Warning.text[readS4_Prompts.outindex] := readS4_Warnings.theemessage;
END_ACTION

ACTION actS5:
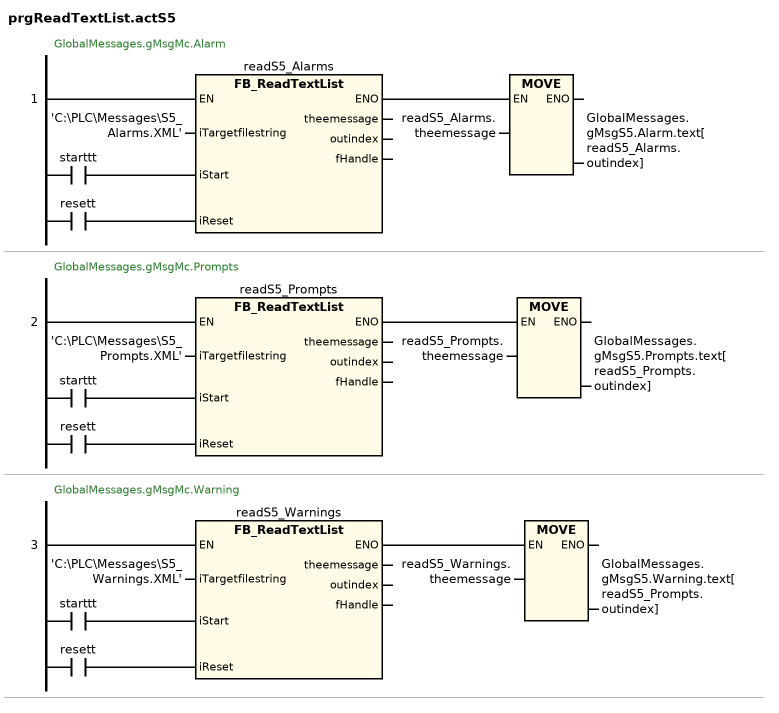
// NETWORK 1
// GlobalMessages.gMsgMc.Alarm
readS5_Alarms(iTargetfilestring := 'C:\PLC\Messages\S5_Alarms.XML', iStart := starttt, iReset := resett); // FB_ReadTextList
GlobalMessages.gMsgS5.Alarm.text[readS5_Alarms.outindex] := readS5_Alarms.theemessage;

// NETWORK 2
// GlobalMessages.gMsgMc.Prompts
readS5_Prompts(iTargetfilestring := 'C:\PLC\Messages\S5_Prompts.XML', iStart := starttt, iReset := resett); // FB_ReadTextList
GlobalMessages.gMsgS5.Prompts.text[readS5_Prompts.outindex] := readS5_Prompts.theemessage;

// NETWORK 3
// GlobalMessages.gMsgMc.Warning
readS5_Warnings(iTargetfilestring := 'C:\PLC\Messages\S5_Warnings.XML', iStart := starttt, iReset := resett); // FB_ReadTextList
GlobalMessages.gMsgS5.Warning.text[readS5_Prompts.outindex] := readS5_Warnings.theemessage;
END_ACTION

ACTION actS6:
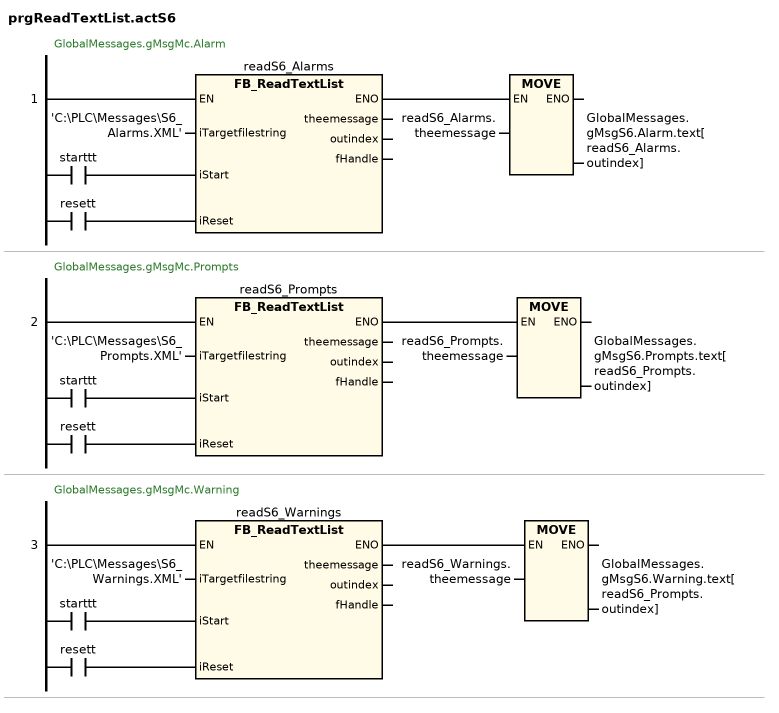
// NETWORK 1
// GlobalMessages.gMsgMc.Alarm
readS6_Alarms(iTargetfilestring := 'C:\PLC\Messages\S6_Alarms.XML', iStart := starttt, iReset := resett); // FB_ReadTextList
GlobalMessages.gMsgS6.Alarm.text[readS6_Alarms.outindex] := readS6_Alarms.theemessage;

// NETWORK 2
// GlobalMessages.gMsgMc.Prompts
readS6_Prompts(iTargetfilestring := 'C:\PLC\Messages\S6_Prompts.XML', iStart := starttt, iReset := resett); // FB_ReadTextList
GlobalMessages.gMsgS6.Prompts.text[readS6_Prompts.outindex] := readS6_Prompts.theemessage;

// NETWORK 3
// GlobalMessages.gMsgMc.Warning
readS6_Warnings(iTargetfilestring := 'C:\PLC\Messages\S6_Warnings.XML', iStart := starttt, iReset := resett); // FB_ReadTextList
GlobalMessages.gMsgS6.Warning.text[readS6_Prompts.outindex] := readS6_Warnings.theemessage;
END_ACTION

END_PROGRAM

// ---- HMI1/Logic/FB_ReadTextList.TcPOU
FUNCTION_BLOCK FB_ReadTextList
VAR_INPUT
	iTargetfilestring:STRING(255):= 'C:\PLC\Messages\FileName.XML'; // 'C:\PLC\Messages\Mc_Alarms.XML'
	iStart: BOOL;
	iReset: BOOL;


END_VAR
VAR_OUTPUT
	theemessage:string(255);
	outindex:INT;
	

END_VAR

VAR_OUTPUT
fHandle:UINT;
END_VAR


VAR
	
	openfileee: FB_FileOpen;
	openfileee2: FB_FileOpen; //used for nulling
	openTheFile: BOOL;
	gettaTheFile: FB_FileGets;
	gettaTheFile2: FB_FileGets; //used for nulling
	readatheFile: BOOL;
	textListNameLocation: INT;
	findText: FB_FindTextIndexNum;
	findLangText: FB_FindTextLangText;
	examplestring: STRING(255);
	tResetFunc: BOOL;
	fileNumber: UINT;
	fileisEOF: BOOL;
	closeatheFile: FB_FileClose;
	IsCorrectLineForText: INT;
	isCorrectLine: BOOL;
	
	startProc:R_Trig; //start reading from file
	closefiletrig:R_TRIG;
	inputreset:R_TRIG;
	readathefileOSR:R_TRIG;
	
	lineIsValidOSR:R_TRIG;
	tResetFunOSR:R_TRIG;
	
	
END_VAR

//start OSR
startProc(CLK := iStart);
openTheFile := startProc.Q;

//open file to get the hfile handle
openfileee(	sNetId		:=,
			sPathName	:=iTargetfilestring,
			nMode		:=FOPEN_MODEREAD,
			ePath		:=PATH_GENERIC,
			bExecute	:=openTheFile,
			tTimeout	:=T#1S
			);
//:= openfileee.bBusy
//:= openfileee.bError
//:= openfileee.nErrId
fileNumber := openfileee.hFile; 

//put handle outside for diagnostics
fHandle := fileNumber;

//close file on complete of the above scan
IF (findText.qIndexNum > GlobalMessages.gNumMessagesPerType) OR tResetFunc THEN
	closeatheFile.bExecute := TRUE;
	ELSE
	closeatheFile.bExecute := FALSE;
END_IF

closeatheFile	(	sNetId		:=,
					hFile		:=fileNumber,
					bExecute	:=,
					tTimeout	:=T#1S
					);
					
//:=	closeatheFile.bBusy
//:=	closeatheFile.bError
//:=	closeatheFile.nErrId 


//OSRs for resetting function
closefiletrig(		CLK :=	closeatheFile.bBusy);
inputreset(			CLK	:=	iReset);

IF closefiletrig.Q OR inputreset.Q THEN
	fileNumber 	:= 0;
	tResetFunc	:= TRUE;
	ELSE
	tResetFunc	:= FALSE;	
END_IF

//read each line of file
IF NOT tResetFunc THEN
	gettaTheFile(	sNetId	:=,
					hFile	:=	fileNumber,
					bExecute:= readatheFile OR tResetFunc,
					tTimeout:= T#1S
					);
	
	fileisEOF := gettaTheFile.bEOF;
END_IF

//on reset, clear file number, can't remove the bEOF since beckhoff can't write to an output
IF tResetFunc THEN
	fileNumber 	:= 0;
	openTheFile	:= FALSE;
	fileisEOF	:= FALSE;
END_IF

//clear instance memory
//not sure if it works, but I would like to think that clearing out the data is the right thing to reset the STAT and output bits
IF tResetFunc THEN
	openfileee := openfileee2;
	gettaTheFile := gettaTheFile2;
END_IF

//check if file opened
IF 	fileNumber > 1 AND 
	NOT tResetFunc AND 
	NOT fileisEOF 
	AND System.oneMilliSecond
	THEN
		readatheFile := TRUE;
	ELSE
		readatheFile := FALSE;
END_IF
//find the integer of the textlist from the XML
findText(iText	:= gettaTheFile.sLine);

//:=	findtext.qIndexNum
//:=	findtext.qLineIsValid
	
//increment XML counter for next usage of text, default text or translated text that apears below
readathefileOSR(CLK:=readatheFile);
IF readathefileOSR.Q THEN
	IsCorrectLineForText := IsCorrectLineForText + 1;
END_IF


//reset XML counter
lineIsValidOSR	(CLK	:= findText.qLineIsValid);
tResetFunOSR	(CLK	:= tResetFunc);

IF lineIsValidOSR.Q OR tResetFunOSR.Q THEN
	IsCorrectLineForText := 0;
END_IF

//check line diffrence between number line and text line
//SET LANGUAGE FOR READING FROM TEXT LISTS HERE ¬
IF IsCorrectLineForText = LanguageLocation.DefaultLanguage THEN
	isCorrectLine := TRUE;
	ELSE
	isCorrectLine := FALSE;
END_IF

//-find language text in default language
//-find in each call each further translated text in <v>German</v> strings in the XML
findLangText(iText:=gettaTheFile.sLine);


//default text entry
IF isCorrectLine AND findLangText.qIsValidString THEN
	examplestring := findLangText.qTextidline3;
END_IF


//extended text for other languages, other than the default one (first entry in beckhoff)
IF isCorrectLine AND findLangText.qIsValidExtendedString THEN
	examplestring := findLangText.qExtendedTextline;
END_IF

//write data into index
IF isCorrectLine AND
	findLangText.qIsValidExtendedString OR findLangText.qIsValidString THEN
	theemessage := examplestring;
	outindex := findText.qIndexNum;
END_IF

END_FUNCTION_BLOCK

// ---- HMI1/Logic/FB_FindTextIndexNum.TcPOU
FUNCTION_BLOCK FB_FindTextIndexNum
VAR_INPUT
	iText:T_MaxString; //input text string to find text in
END_VAR
VAR_OUTPUT
	qIndexNum: INT; //index number of string
	qLineIsValid: BOOL; //TRUE if the line valid to be processed?
END_VAR
VAR
	textidNameLocation: INT;
	textIDlocname: STRING(255);
	isTextIDLinee: BOOL;
	textidline: INT;
	textIDnameLefted: STRING(255);
	textidline2: INT;
	textlen: INT;
	textidline3: STRING(255);
	indexIsInt: BOOL;
END_VAR
//theme:ZmgvZTlLAsU

//find text entry name
//'              <v n="TextID">"0"</v>$N' '              <v n="TextDefault">"Example alarm for Mc_Alarms"</v>$N'
textidNameLocation	:=		FIND	(STR1:=iText, 			STR2:= 'TextID');

//finds,
//'Mc_Alarms" Id="{4f6'
IF textidNameLocation >= 1 THEN
	textIDlocname	:=	iText;
	isTextIDLinee	:=	TRUE;
	ELSE
	isTextIDLinee	:=	FALSE;
END_IF

//find end OF line, converts,
//'TextID">"0"</v>$N'
//-3
//to
//'TextID">"0"'
textidline	:= 				FIND	(STR1:=textIDlocname,	STR2:='"</v>');
textIDnameLefted :=			LEFT	(STR:=textIDlocname, 	SIZE:=textidline -1);

IF isTextIDLinee THEN
	textidline2	:=			FIND	(STR1:=textIDnameLefted,STR2:='">"');
	textlen		:=			LEN		(STR:=textIDnameLefted);
	textidline3 :=			RIGHT	(STR:=textIDnameLefted, SIZE:= textlen - textidline2 - 2);
END_IF

qIndexNum := STRING_TO_INT(textidline3);

IF qIndexNum >= -1 THEN 
	indexIsInt := TRUE;
ELSE
	indexIsInt := FALSE;
END_IF

//output if line is valid
IF isTextIDLinee AND  indexIsInt THEN
	qLineIsValid := TRUE;
	ELSE
	qLineIsValid := FALSE;
END_IF

END_FUNCTION_BLOCK

// ---- HMI1/Logic/FB_FindTextLangText.TcPOU
FUNCTION_BLOCK FB_FindTextLangText
VAR_INPUT
		iText:T_MaxString;
END_VAR
VAR_OUTPUT
		qTextidline3: STRING(255);
		qIsValidString: BOOL;
		qExtendedTextline: STRING(255);
		qIsValidExtendedString: BOOL;
END_VAR
VAR
		textidNameLocation: INT;
		textIDlocname: STRING(255);
		isTextIDLinee: BOOL;
		textidline: INT;
		textIDnameLefted: STRING(255);
		textidline2: INT;
		textlen: INT;

		textlencheck: INT;
		textmencheckvalid: BOOL;
		isExtendedLang: BOOL;
		vLocation: INT;
		strExtended: STRING(255);
		lenstrExtneded: INT;
		endVlocation: INT;
		isExtendedLangendV: BOOL;
		resultstrExtended: STRING(255);
END_VAR
//theme:EDn-ZLMZpzA

//find text entry name
//'              <v n="TextDefault">"Example alarm for Mc_Alarms"</v>$N'
textidNameLocation := FIND(STR1:= iText, STR2:='TextDefault');

IF textidNameLocation >= 1 THEN
	textIDlocname := iText;
	isTextIDLinee := TRUE;
	ELSE
	isTextIDLinee := FALSE;
END_IF

//find end of line, converts,
//'              <v n="TextDefault">"Example alarm for Mc_Alarms"</v>$N'
textidline := FIND			(STR1:= textIDlocname, STR2:='"</v>');
textIDnameLefted := LEFT	(STR:= textIDlocname, SIZE:= textidline - 1);

//">" format right of the integer
//"TextDefault">"
IF isTextIDLinee THEN
	textidline2 := FIND		(STR1:= textIDnameLefted, STR2:='"TextDefault">"');
	textlen := LEN			(STR:= textIDnameLefted);
	qTextidline3 := RIGHT	(STR:= textIDnameLefted, SIZE:= textlen - textidline2 - 14);
END_IF

//check if string is a string with a len check >1
textlencheck := LEN(qTextidline3);
IF textlencheck > 1 THEN
	textmencheckvalid := TRUE;
	ELSE
	textmencheckvalid := FALSE;
END_IF

IF isTextIDLinee AND textmencheckvalid THEN
	qIsValidString := TRUE;
	ELSE
	qIsValidString := FALSE;
END_IF

//logic #2, determine presense of 
//<v>german 0</v> XML of <v>
vLocation :=					FIND(STR1:=iText, STR2:= '<v>');
IF vLocation > 1 THEN
	isExtendedLang := TRUE;
	ELSE
	isExtendedLang := FALSE;
END_IF

IF isExtendedLang THEN
	lenstrExtneded := LEN		(STR:=iText);
	strExtended := RIGHT		(STR:= iText,SIZE:= lenstrExtneded - vLocation - 2);
END_IF

//logic #2, determine presense of 
//</v>
//terminator for /v
IF isExtendedLang THEN
	endVlocation := FIND		(STR1:=strExtended, STR2:= '</v>');
	IF endVlocation > 1 THEN
		isExtendedLangendV := TRUE;
		ELSE
		isExtendedLangendV := FALSE;
	END_IF
END_IF

//'german 0</v>$N'
IF isExtendedLangendV AND isExtendedLang THEN
	resultstrExtended := LEFT	(STR:=strExtended, SIZE:= endVlocation - 1);
END_IF

//'german 1'
IF	isExtendedLangendV AND isExtendedLang THEN
	qExtendedTextline := resultstrExtended;
	qIsValidExtendedString := TRUE;
	ELSE
	qIsValidExtendedString := FALSE;
END_IF

END_FUNCTION_BLOCK

// ---- HMI1/Logic/prgHMILanguage.TcPOU
PROGRAM prgHMILanguage
VAR
	tTrueLangIndex: UINT;
	tSizeOfLangRow: UINT;
	tSizeOfLangRowButtons: UINT;
	tStationNumberIndexLang: UINT;
	tScreenElementsPerPageLang: UINT;
	tNumElementsPerScreen: UINT;
	retval: UDINT;
	nextPage: R_TRIG;
	PrevPage: R_TRIG;
END_VAR

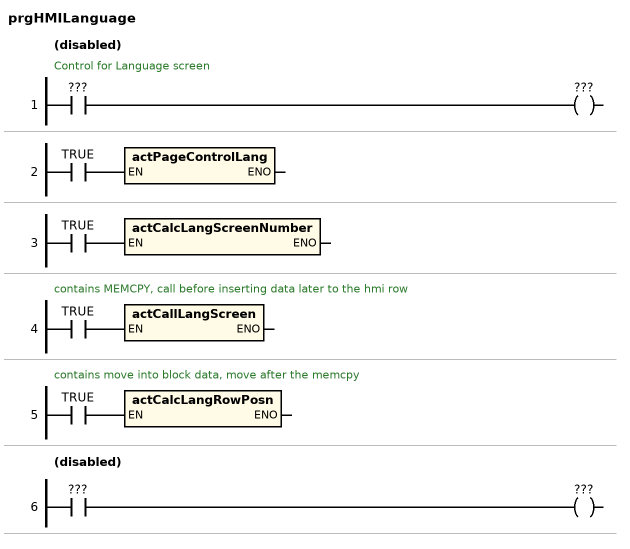
// NETWORK 1 (disabled)
// Control for Language screen
// ??? := ???;

// NETWORK 2
actPageControlLang();

// NETWORK 3
actCalcLangScreenNumber();

// NETWORK 4
// contains MEMCPY, call before inserting data later to the hmi row
actCallLangScreen();

// NETWORK 5
// contains move into block data, move after the memcpy
actCalcLangRowPosn();

// NETWORK 6 (disabled)
// ??? := ???;

ACTION actCalcLangRowPosn:
//calculate station index for pages
tTrueLangIndex :=	tStationNumberIndexLang +
					(tScreenElementsPerPageLang * gHMIData.gActiveLangPageNumber) -  tScreenElementsPerPageLang;
					
//calculate offset for row x
gHMIData.gLangRowElementOffset[1] :=	tTrueLangIndex + 
										(gHMIDataConst.gNumberElementsPerRow * 1) - gHMIDataConst.gNumberElementsPerRow;

gHMIData.gLangRowElementOffset[2] :=	tTrueLangIndex + 
										(gHMIDataConst.gNumberElementsPerRow * 2) - gHMIDataConst.gNumberElementsPerRow;

gHMIData.gLangRowElementOffset[3] :=	tTrueLangIndex + 
										(gHMIDataConst.gNumberElementsPerRow * 3) - gHMIDataConst.gNumberElementsPerRow;

gHMIData.gLangRowElementOffset[4] :=	tTrueLangIndex + 
										(gHMIDataConst.gNumberElementsPerRow * 4) - gHMIDataConst.gNumberElementsPerRow;

gHMIData.gLangRowElementOffset[5] :=	tTrueLangIndex + 
										(gHMIDataConst.gNumberElementsPerRow * 5) - gHMIDataConst.gNumberElementsPerRow;

gHMIData.gLangRowElementOffset[6] :=	tTrueLangIndex + 
										(gHMIDataConst.gNumberElementsPerRow * 6) - gHMIDataConst.gNumberElementsPerRow;
				
//move to global to be picked up by each row					
gHMIData.gLangRows.gMotionRow1.IndexLocation := gHMIData.gLangRowElementOffset[1];
gHMIData.gLangRows.gMotionRow2.IndexLocation := gHMIData.gLangRowElementOffset[2];
gHMIData.gLangRows.gMotionRow3.IndexLocation := gHMIData.gLangRowElementOffset[3];
gHMIData.gLangRows.gMotionRow4.IndexLocation := gHMIData.gLangRowElementOffset[4];
gHMIData.gLangRows.gMotionRow5.IndexLocation := gHMIData.gLangRowElementOffset[5];
gHMIData.gLangRows.gMotionRow6.IndexLocation := gHMIData.gLangRowElementOffset[6];
END_ACTION

ACTION actCalcLangScreenNumber:
//create number for station
tStationNumberIndexLang	:= 1 * 10000; //declare math for now


//calculate number of elements per screen
tNumElementsPerScreen	:= gHMIDataConst.gNumberRowsPerPage * gHMIDataConst.gNumberElementsPerRow;

//calculate screen per page index
tScreenElementsPerPageLang := tNumElementsPerScreen * 1; //declare math for future use
END_ACTION

ACTION actCallLangScreen:
//calculate byte offset - motions
tSizeOfLangRow := gHMIData.gActivePageNumber * SIZEOF(gHMIData.gLangRows); //for pointer use
tSizeOfLangRow := tSizeOfLangRow - SIZEOF(gHMIData.gLangRows);

//calculate byte offset - buttons
tSizeOfLangRowButtons := gHMIData.gActivePageNumber * SIZEOF(gHMIData.gLangButtons);
tSizeOfLangRowButtons := tSizeOfLangRowButtons - SIZEOF(gHMIData.gLangButtons);

//move data based on station and page number
//Move feedback indicator data
//Move Button BOOL state back adr(S1_Global.MotionRow)
MEMCPY(	destAddr	:= ADR(gHMIData.gLangRows),
		srcAddr		:= ADR(Mc_Global.LangRow) + tSizeOfLangRow,
		n			:= SIZEOF(gHMIData.gLangRows)
		);

MEMCPY(	destAddr	:= ADR(Mc_Global.LangRowBtn) + tSizeOfLangRowButtons,
		srcAddr		:= ADR(gHMIData.gLangButtons),
		n			:= sizeof(gHMIData.gLangButtons)
		);
END_ACTION

ACTION actPageControlLang:
//next page
nextPage(CLK	:= gHMIButtons.btnNextPage);
IF nextPage.Q THEN
	gHMIData.gActiveLangPageNumber	:=	gHMIData.gActiveLangPageNumber + 1;
END_IF

//previous page
PrevPage(CLK	:= gHMIButtons.btnPrevPage);
IF PrevPage.Q THEN
	gHMIData.gActiveLangPageNumber := gHMIData.gActiveLangPageNumber - 1;
END_IF



//apply limits
IF gHMIData.gActiveLangPageNumber < 1 THEN
	gHMIData.gActiveLangPageNumber := 1;
END_IF
	
IF gHMIData.gActiveLangPageNumber > gHMIData.gMaxPageNumberLang THEN
	gHMIData.gActiveLangPageNumber := 1;
END_IF

gHMIData.gMaxPageNumberLang := Mc_Global.Data.NumberOfPages;
END_ACTION

END_PROGRAM

// ---- HMI1/Logic/prgHMIaxis.TcPOU
PROGRAM prgHMIaxis
VAR
	
	i: UINT;
END_VAR

//logic for HMI diag screens for axis

//assign text for diag screen
FOR i := 1 TO Axis.gNumAxisInSystem DO
	//populate dropdown box
	driveGlobals.tAxisList[i] := Axis.axisPresent[i].AxisName;
END_FOR

//assign nc info to HMI nc info
CASE driveGlobals.hmiAxisSel OF
	1:	driveGlobals.hmiAxis :=driveGlobals.ncAxis1;
	2:	driveGlobals.hmiAxis :=driveGlobals.ncAxis2;
	3:	driveGlobals.hmiAxis :=driveGlobals.ncAxis3;
	4:	driveGlobals.hmiAxis :=driveGlobals.ncAxis4;
	5:	driveGlobals.hmiAxis :=driveGlobals.ncAxis5;
	6:	driveGlobals.hmiAxis :=driveGlobals.ncAxis6;
	7:	driveGlobals.hmiAxis :=driveGlobals.ncAxis7;
	8:	driveGlobals.hmiAxis :=driveGlobals.ncAxis8;	
END_CASE

END_PROGRAM

// ---- HMI1/Logic/prgModeRows.TcPOU
PROGRAM prgModeRows
VAR
	
ModeRow1:FB_HMI_Control_NoGroupRef;
ModeRow2:FB_HMI_Control_NoGroupRef;
ModeRow3:FB_HMI_Control_NoGroupRef;
ModeRow4:FB_HMI_Control_NoGroupRef;
ModeRow5:FB_HMI_Control_NoGroupRef;
ModeRow6:FB_HMI_Control_NoGroupRef;
ModeRow7:FB_HMI_Control_NoGroupRef;
ModeRow8:FB_HMI_Control_NoGroupRef;
ModeRow9:FB_HMI_Control_NoGroupRef;

ModeRowsStn: typeStation;
	tNumRows: UINT;
END_VAR

VAR_INPUT
	MotionRowLocation: typeMotionRow;
END_VAR

//theme:VNPKlVq0z2Y

//zero indexing code
tNumRows := 0;

//clear HMI row for manual insertion
gModeAlternate.gModeRows.gMotionRow1.IndexLocation := 0;
gModeAlternate.gModeRows.gMotionRow2.IndexLocation := 20;
gModeAlternate.gModeRows.gMotionRow3.IndexLocation := 40;
gModeAlternate.gModeRows.gMotionRow4.IndexLocation := 60;
gModeAlternate.gModeRows.gMotionRow5.IndexLocation := 80;
gModeAlternate.gModeRows.gMotionRow6.IndexLocation := 100;
gModeAlternate.gModeRows.gMotionRow7.IndexLocation := 120;
gModeAlternate.gModeRows.gMotionRow8.IndexLocation := 140;
gModeAlternate.gModeRows.gMotionRow9.IndexLocation := 160;

//call the rows
actcallRows();

ACTION actCallRows:
//theme:ETfiUYij5UE
//hard code location and address for special case of alternate motion row use for mode


//motion row 1, Power ON/OFF
ModeRow1	(	iStationNumber		:=1,
				iRowNumber			:=1,
				iAdvanceLimit		:=Mc_Global.PowerOnFdbk,
				iReturnLimit		:=NOT Mc_Global.PowerOnFdbk,
				iAdvanceCoil		:=gModeAlternate.gModeButtons.gMotionRow1btn.btnAdvance,
				iReturnCoil			:=gModeAlternate.gModeButtons.gMotionRow1btn.btnReturn,
				iAdvanceTime		:=,
				iReturnTime			:=,
				iAdvanceInterlock	:=,
				iReturnInterlock	:=,
				iAdvancePrompt		:=,
				iReturnPrompt		:=,
				iConfig				:=RowConfig.FullRowNoVal,
				iAdvanceNumber		:=0,
				iReturnNumber		:=0,
				iUnits				:='',
				iPosn				:='',
				NumRows				:=tNumRows,
				MotionRowLocation	:=gModeAlternate.gModeRows.gMotionRow1,
				MotionRowBtnLocation:=gModeAlternate.gModeButtons.gMotionRow1btn
				);

//manually set row number for textlist offset				
gModeAlternate.gModeRows.gMotionRow1.IndexLocation := gModeAlternate.gModeRows.gMotionRow1.IndexLocation + 10000;			


//motion row 2, Auto / Manual
ModeRow2	(	iStationNumber		:=1,
				iRowNumber			:=2,
				iAdvanceLimit		:=gHMIButtons.btnFdbk.btn00Fdbk,
				iReturnLimit		:=gHMIButtons.btnFdbk.btn01Fdbk,
				iAdvanceCoil		:=gModeAlternate.gModeButtons.gMotionRow2btn.btnAdvance,
				iReturnCoil			:=gModeAlternate.gModeButtons.gMotionRow2btn.btnReturn,
				iAdvanceTime		:=,
				iReturnTime			:=,
				iAdvanceInterlock	:=,
				iReturnInterlock	:=,
				iAdvancePrompt		:=,
				iReturnPrompt		:=,
				iConfig				:=RowConfig.FullRowNoVal,
				iAdvanceNumber		:=0,
				iReturnNumber		:=0,
				iUnits				:='',
				iPosn				:='',
				NumRows				:=tNumRows,
				MotionRowLocation	:=gModeAlternate.gModeRows.gMotionRow2,
				MotionRowBtnLocation:=gModeAlternate.gModeButtons.gMotionRow2btn
				);
				
				
//manually set row number for textlist offset				
gModeAlternate.gModeRows.gMotionRow2.IndexLocation := gModeAlternate.gModeRows.gMotionRow2.IndexLocation + 10000;			


